ABB RobotStudio station: Celda_Paletizado_20220202-004534.rsstn

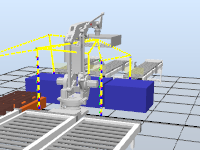
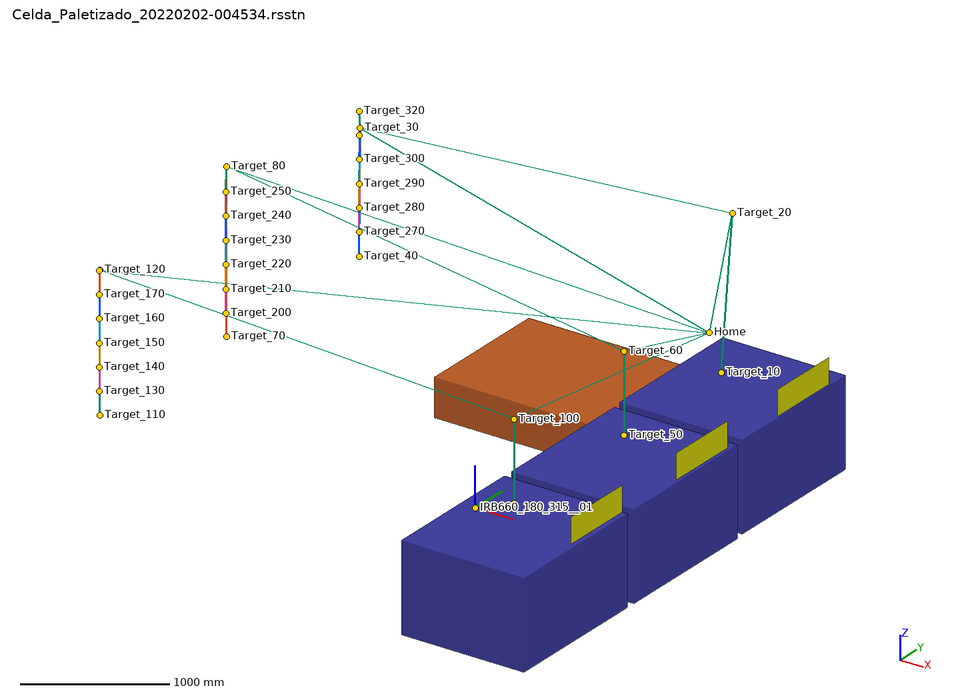
[picture v1: parts stored in the station drawn from their meshes, with robot base, taught points and paths (robot models come from the ABB library and are not in the file)]
Station Celda_Paletizado (saved by RobotStudio 21.4.9700.0)
Controller IRB660_180_315
  mechanical unit ROB_1: IRB660_180_315__01, 6 joints, base frame (0, 0, 0) mm
Layout (positions relative to the parent item):
  - IRB660_180_315__01 [mechanism, from Robots\IRB660_180_315__01.rslib] at (0, 0, 0) mm; joint values [0, 0.0198, -0.194, 0] (rad or m)
  - 600_guide [part, from Equipment\Conveyor Guide 600.rslib] at (4720, 275, 0) mm, rotated rx 0 ry 0 rz 180 deg
  - 600_guide_2 [part, from Equipment\Conveyor Guide 600.rslib] at (4720, 1475, 0) mm, rotated rx 0 ry 0 rz 180 deg
  - 600_guide_3 [part, from Equipment\Conveyor Guide 600.rslib] at (4720, -900, 0) mm, rotated rx 0 ry 0 rz 180 deg
  - 1200_4000_h2_2 [part, from Equipment\Conveyor 1200 4000 h2.rslib] at (-1500, -1000, 0) mm, rotated rx 0 ry 0 rz 180 deg
  - 1200_4000_h2_3 [part, from Equipment\Conveyor 1200 4000 h2.rslib] at (-1500, 2000, 0) mm, rotated rx 0 ry 0 rz 180 deg
  - 1200_4000_h2_4 [part, from Equipment\Conveyor 1200 4000 h2.rslib] at (-1500, 500, 0) mm, rotated rx 0 ry 0 rz 180 deg
  - 1200_4800_h2_2 [part, from Equipment\Conveyor 1200 4800 h2.rslib] at (-6865.5, 2181.45, 0) mm, rotated rx 0 ry 0 rz -90 deg
  - Pieza_1 [part] at (-5740.3, -4363.37, 0) mm, rotated rx 0 ry 0 rz 90 deg, size 1600 x 1000 x 355 mm
  - wraping_1 [part] at (-6239.59, -3461.03, 366.67) mm, rotated rx 0 ry 0 rz -90 deg, size 2370 x 1393.7 x 2100 mm
  - wraping_2 [part] at (-6238.99, -3463.39, 358.4) mm, rotated rx 0 ry 0 rz -90 deg, size 1400 x 1393.6 x 350 mm
  - wraping_3 [part] at (-6242.7, -3445.47, -111.4) mm, rotated rx 90 ry 0 rz -90 deg, size 323.7 x 500 x 658.2 mm
  - Pieza_4 [part] at (-1012.61, 969.79, 0) mm, size 1300 x 1100 x 300 mm
  - Pieza_6 [part] at (689.01, 695.64, 0) mm, size 1000 x 1200 x 700 mm
  - Pieza_7 [part] at (702.6, -1863.75, 0) mm, size 1000 x 1200 x 700 mm
  - Pieza_8 [part] at (703.57, -585.32, 0) mm, size 1000 x 1200 x 700 mm
  - Mi_mecanismo [mechanism] at (1910, 0, 2093) mm; joint values [0, 0] (rad or m)
      TCP Mi_mecanismo_1 at (1.05, 425.12, 399.16) mm, rotated rx 90 ry 0 rz 180 deg
      links: L1, L2, L3
  - Euro Pallet [graphiccomponentgroup, from Equipment\Euro Pallet.rslib] at (223.77, 1878.53, 297.19) mm, rotated rx 0 ry 0 rz 180 deg
    - Body 1 [part, from Equipment\Euro Pallet.rslib]
  - Euro Pallet_2 [graphiccomponentgroup, from Equipment\Euro Pallet.rslib] at (-1565.85, 821.96, 434.35) mm, rotated rx 0 ry 0 rz 90 deg
    - Body 1 [part, from Equipment\Euro Pallet.rslib]
  - Pieza_19 [part] at (1027.44, -3056.32, 715) mm, rotated rx 0 ry 0 rz 90 deg, size 425 x 325 x 180 mm
  - Pequeño [smart component] at (5282.75, -525.09, 765.47) mm
      signals: DI Start, DI Cinta, DI Coger, DI Soltar, DO Sensor1, DO Recoger_peq
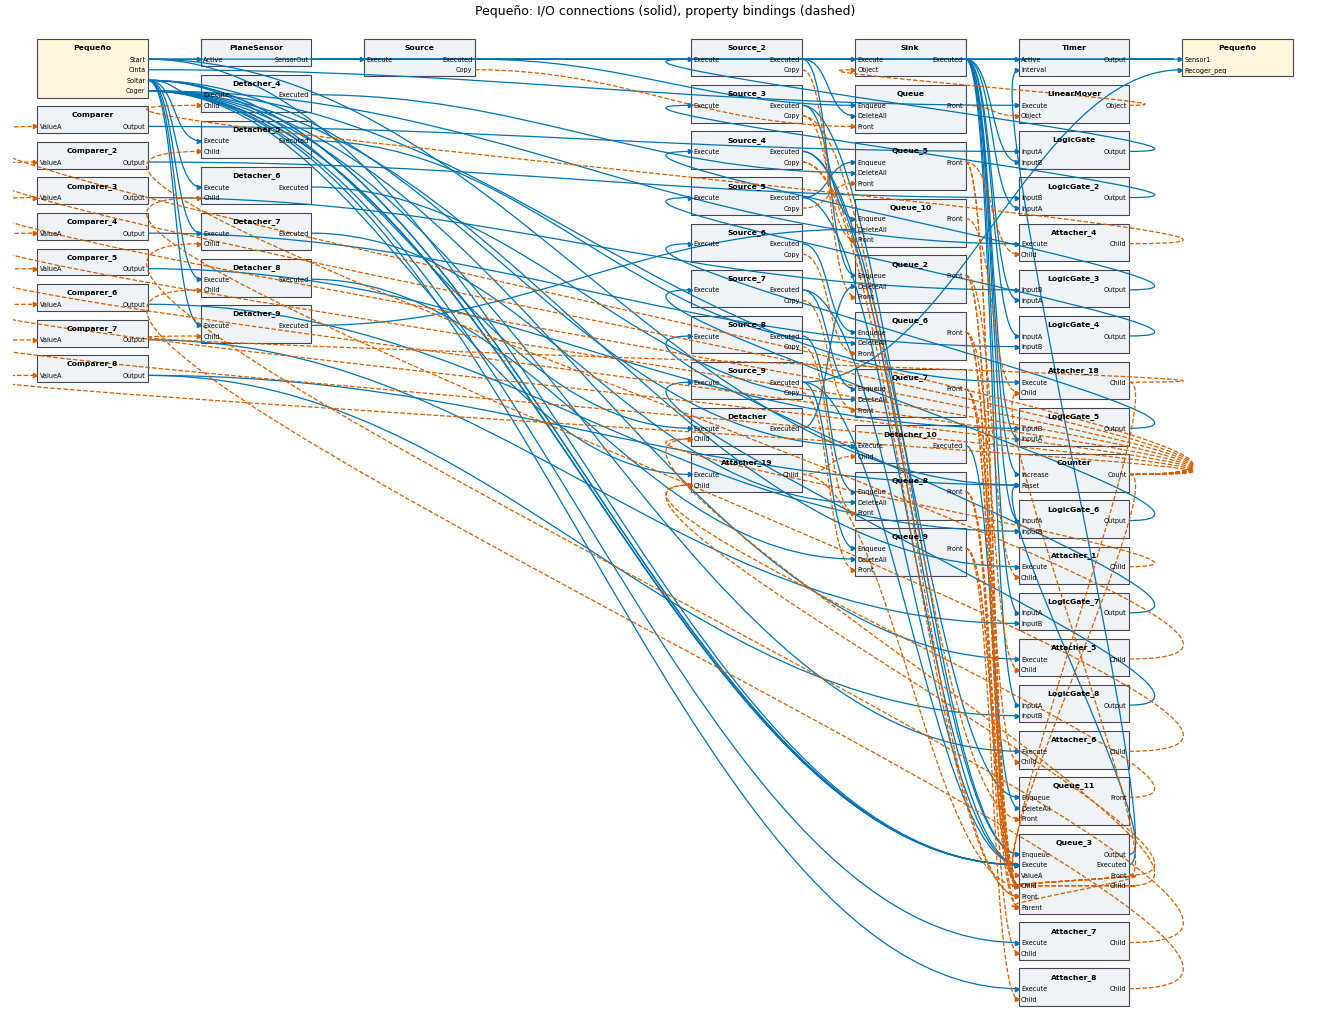
      connections:
        Pequeño.Start -> Timer.Active
        Timer.Output -> Source.Execute
        Source.Executed -> Queue.Enqueue
        Pequeño.Cinta -> LinearMover.Execute
        Pequeño.Start -> PlaneSensor.Active
        PlaneSensor.SensorOut -> Sink.Execute
        Source_2.Executed -> Queue_2.Enqueue
        Sink.Executed -> Counter.Increase
        LogicGate.Output -> Source_2.Execute
        Comparer.Output -> LogicGate.InputA
        Sink.Executed -> LogicGate.InputB
        Comparer_2.Output -> LogicGate_2.InputB
        Sink.Executed -> LogicGate_2.InputA
        LogicGate_2.Output -> Source_3.Execute
        Source_3.Executed -> Queue_3.Enqueue
        PlaneSensor.SensorOut -> Pequeño.Sensor1
        Comparer_3.Output -> LogicGate_3.InputB
        LogicGate_3.Output -> Source_4.Execute
        Sink.Executed -> LogicGate_3.InputA
        Source_4.Executed -> Queue_4.Enqueue
        Sink.Executed -> LogicGate_4.InputA
        Comparer_4.Output -> LogicGate_4.InputB
        LogicGate_4.Output -> Source_5.Execute
        Source_5.Executed -> Queue_5.Enqueue
        Comparer_5.Output -> LogicGate_5.InputB
        Sink.Executed -> LogicGate_5.InputA
        LogicGate_5.Output -> Source_6.Execute
        Source_6.Executed -> Queue_6.Enqueue
        Sink.Executed -> LogicGate_6.InputA
        Comparer_6.Output -> LogicGate_6.InputB
        LogicGate_6.Output -> Source_7.Execute
        Source_7.Executed -> Queue_7.Enqueue
        Sink.Executed -> LogicGate_7.InputA
        Comparer_7.Output -> LogicGate_7.InputB
        LogicGate_7.Output -> Source_8.Execute
        Source_8.Executed -> Queue_8.Enqueue
        Sink.Executed -> LogicGate_8.InputA
        Comparer_8.Output -> LogicGate_8.InputB
        LogicGate_8.Output -> Source_9.Execute
        Source_9.Executed -> Queue_9.Enqueue
        Comparer_9.Output -> Counter.Reset
        Comparer_8.Output -> Counter.Reset
        Pequeño.Start -> Counter.Reset
        Pequeño.Soltar -> Detacher.Execute
        Source_9.Executed -> Pequeño.Recoger_peq
        Pequeño.Coger -> Attacher.Execute
        Source_7.Executed -> Attacher_6.Execute
        Source_5.Executed -> Attacher_5.Execute
        Source_9.Executed -> Attacher_7.Execute
        Pequeño.Coger -> Attacher_1.Execute
        Pequeño.Coger -> Attacher_2.Execute
        Pequeño.Coger -> Attacher_3.Execute
        Pequeño.Coger -> Attacher_4.Execute
        Pequeño.Coger -> Attacher_5.Execute
        Pequeño.Coger -> Attacher_6.Execute
        Pequeño.Coger -> Attacher_7.Execute
        Pequeño.Coger -> Attacher_8.Execute
        Pequeño.Soltar -> Detacher_2.Execute
        Pequeño.Soltar -> Detacher_3.Execute
        Pequeño.Soltar -> Detacher_4.Execute
        Pequeño.Soltar -> Detacher_5.Execute
        Pequeño.Soltar -> Detacher_6.Execute
        Pequeño.Soltar -> Detacher_7.Execute
        Pequeño.Soltar -> Detacher_8.Execute
        Pequeño.Coger -> Attacher_18.Execute
        Pequeño.Coger -> Attacher_19.Execute
        Pequeño.Soltar -> Detacher_9.Execute
        Pequeño.Soltar -> Detacher_10.Execute
        Source_4.Executed -> Queue_11.Enqueue
        Source_3.Executed -> Queue_10.Enqueue
        Source_2.Executed -> Queue.DeleteAll
        Detacher.Executed -> Queue_2.DeleteAll
        Detacher_9.Executed -> Queue_10.DeleteAll
        Detacher_10.Executed -> Queue_11.DeleteAll
        Detacher_4.Executed -> Queue_5.DeleteAll
        Detacher_5.Executed -> Queue_6.DeleteAll
        Detacher_6.Executed -> Queue_7.DeleteAll
        Detacher_7.Executed -> Queue_8.DeleteAll
        Detacher_8.Executed -> Queue_9.DeleteAll
        Random.Executed -> Timer.Interval
        Pequeño.Start -> Random.Execute
        Source.Copy => Queue.Front
        Queue.Front => LinearMover.Object
        LinearMover.Object => Sink.Object
        Counter.Count => Comparer.ValueA
        Counter.Count => Comparer_2.ValueA
        Counter.Count => Comparer_3.ValueA
        Counter.Count => Comparer_4.ValueA
        Counter.Count => Comparer_5.ValueA
        Counter.Count => Comparer_6.ValueA
        Counter.Count => Comparer_7.ValueA
        Counter.Count => Comparer_8.ValueA
        Counter.Count => Comparer_9.ValueA
        Queue_2.Front => Attacher.Child
        Queue_3.Front => Attacher.Child
        Queue_4.Front => Attacher.Child
        Queue_5.Front => Attacher.Child
        Queue_6.Front => Attacher.Child
        Queue_7.Front => Attacher.Child
        Queue_8.Front => Attacher.Child
        Queue_9.Front => Attacher.Child
        Attacher.Child => Detacher.Child
        Source_2.Copy => Queue_2.Front
        Source_3.Copy => Queue_3.Front
        Source_4.Copy => Queue_4.Front
        Source_5.Copy => Queue_5.Front
        Source_6.Copy => Queue_6.Front
        Source_7.Copy => Queue_7.Front
        Source_8.Copy => Queue_8.Front
        Source_9.Copy => Queue_9.Front
        Queue_2.Front => Attacher_3.Child
        Attacher_1.Child => Detacher.Child
        Queue_4.Front => Attacher_5.Parent
        Queue_5.Front => Attacher_5.Child
        Queue_6.Front => Attacher_6.Parent
        Queue_7.Front => Attacher_6.Child
        Queue_8.Front => Attacher_7.Parent
        Queue_9.Front => Attacher_7.Child
        Queue_3.Front => Attacher_2.Child
        Queue_4.Front => Attacher_3.Child
        Queue_5.Front => Attacher_4.Child
        Queue_6.Front => Attacher_5.Child
        Queue_7.Front => Attacher_6.Child
        Queue_8.Front => Attacher_7.Child
        Queue_9.Front => Attacher_8.Child
        Attacher_2.Child => Detacher_2.Child
        Attacher_3.Child => Detacher_3.Child
        Attacher_4.Child => Detacher_4.Child
        Attacher_5.Child => Detacher_5.Child
        Attacher_6.Child => Detacher_6.Child
        Attacher_7.Child => Detacher_7.Child
        Attacher_8.Child => Detacher_8.Child
        Queue_2.Front => Attacher_1.Child
        Queue_3.Front => Attacher_18.Child
        Queue_4.Front => Attacher_19.Child
        Attacher_18.Child => Detacher_2.Child
        Attacher_19.Child => Detacher_3.Child
        Source_4.Copy => Queue_11.Front
        Source_3.Copy => Queue_10.Front
        Queue_10.Front => Attacher_18.Child
        Queue_11.Front => Attacher_19.Child
        Attacher_18.Child => Detacher_9.Child
        Attacher_19.Child => Detacher_10.Child
    - LinearMover [smart component, from Components\LinearMover.rslib]
        properties: Object=(none); Direction=[-0.001 0 0]; Speed=1.5; Reference=Global; ReferenceObject=(none)
    - PlaneSensor [smart component, from Components\PlaneSensor.rslib] at (-3443.45, 1412.3, 72.76) mm, rotated rx 0 ry -90 rz 0 deg
        properties: Origin=[0 0 0]; Axis1=[0.2 0 0]; Axis2=[0 0.6 0]; SensedPart=(none)
      - _sensorPart_ [part], size 200 x 600 x 0 mm
    - Detacher [smart component, from Components\Detacher.rslib]
        properties: Child=(none); KeepPosition=true
    - Queue [smart component, from Components\Queue.rslib]
        properties: Back=(none); Front=(none); Queue=; NumberOfObjects=0
    - Source [smart component, from Components\Source.rslib]
        properties: Source=Pieza_19; Copy=(none); Parent=(none); Position=[4.6 0.975 0.775]; Orientation=[0 0 1.5707963267949]; Transient=true; PhysicsBehavior=0
    - Timer [smart component, from Components\Timer.rslib]
        properties: StartTime=0; Interval=3; Repeat=true; CurrentTime=11.448
    - Sink [smart component, from Components\Sink.rslib]
        properties: Object=(none)
    - Source_2 [smart component, from Components\Source.rslib]
        properties: Source=Pieza_19; Copy=(none); Parent=(none); Position=[1.015 1.47 0.7]; Orientation=[0 0 1.5707963267949]; Transient=false; PhysicsBehavior=0
    - Source_3 [smart component, from Components\Source.rslib]
        properties: Source=Pieza_19; Copy=(none); Parent=(none); Position=[1.345 1.47 0.7]; Orientation=[0 0 1.5707963267949]; Transient=false; PhysicsBehavior=0
    - Source_4 [smart component, from Components\Source.rslib]
        properties: Source=Pieza_19; Copy=(none); Parent=(none); Position=[1.675 1.47 0.7]; Orientation=[0 0 1.5707963267949]; Transient=false; PhysicsBehavior=0
    - Queue_2 [smart component, from Components\Queue.rslib]
        properties: Back=(none); Front=(none); Queue=; NumberOfObjects=0
    - Counter [smart component, from Components\Counter.rslib]
        properties: Count=0
    - LogicGate [smart component, from Components\LogicGate.rslib]
        properties: Operator=AND; Delay=0
    - Comparer [smart component, from Components\Comparer.rslib]
        properties: ValueA=0; Operator===; ValueB=1
    - Comparer_2 [smart component, from Components\Comparer.rslib]
        properties: ValueA=0; Operator===; ValueB=2
    - Comparer_3 [smart component, from Components\Comparer.rslib]
        properties: ValueA=0; Operator===; ValueB=3
    - Comparer_4 [smart component, from Components\Comparer.rslib]
        properties: ValueA=0; Operator===; ValueB=4
    - Comparer_5 [smart component, from Components\Comparer.rslib]
        properties: ValueA=0; Operator===; ValueB=5
    - Comparer_6 [smart component, from Components\Comparer.rslib]
        properties: ValueA=0; Operator===; ValueB=6
    - Comparer_7 [smart component, from Components\Comparer.rslib]
        properties: ValueA=0; Operator===; ValueB=7
    - LogicGate_2 [smart component, from Components\LogicGate.rslib]
        properties: Operator=AND; Delay=0
    - LogicGate_3 [smart component, from Components\LogicGate.rslib]
        properties: Operator=AND; Delay=0
    - LogicGate_4 [smart component, from Components\LogicGate.rslib]
        properties: Operator=AND; Delay=0
    - LogicGate_5 [smart component, from Components\LogicGate.rslib]
        properties: Operator=AND; Delay=0
    - LogicGate_6 [smart component, from Components\LogicGate.rslib]
        properties: Operator=AND; Delay=0
    - LogicGate_7 [smart component, from Components\LogicGate.rslib]
        properties: Operator=AND; Delay=0
    - Queue_5 [smart component, from Components\Queue.rslib]
        properties: Back=(none); Front=(none); Queue=; NumberOfObjects=0
    - Queue_6 [smart component, from Components\Queue.rslib]
        properties: Back=(none); Front=(none); Queue=; NumberOfObjects=0
    - Queue_7 [smart component, from Components\Queue.rslib]
        properties: Back=(none); Front=(none); Queue=; NumberOfObjects=0
    - Queue_8 [smart component, from Components\Queue.rslib]
        properties: Back=(none); Front=(none); Queue=; NumberOfObjects=0
    - Source_5 [smart component, from Components\Source.rslib]
        properties: Source=Pieza_19; Copy=(none); Parent=(none); Position=[0.69 1.14 0.7]; Orientation=[0 0 0]; Transient=false; PhysicsBehavior=0
    - Source_6 [smart component, from Components\Source.rslib]
        properties: Source=Pieza_19; Copy=(none); Parent=(none); Position=[1.255 1.14 0.7]; Orientation=[0 0 0]; Transient=false; PhysicsBehavior=0
    - Source_7 [smart component, from Components\Source.rslib]
        properties: Source=Pieza_19; Copy=(none); Parent=(none); Position=[1.015 0.71 0.7]; Orientation=[0 0 1.5707963267949]; Transient=false; PhysicsBehavior=0
    - Source_8 [smart component, from Components\Source.rslib]
        properties: Source=Pieza_19; Copy=(none); Parent=(none); Position=[1.345 0.71 0.7]; Orientation=[0 0 1.5707963267949]; Transient=false; PhysicsBehavior=0
    - Comparer_8 [smart component, from Components\Comparer.rslib]
        properties: ValueA=0; Operator=>=; ValueB=8
    - Source_9 [smart component, from Components\Source.rslib]
        properties: Source=Pieza_19; Copy=(none); Parent=(none); Position=[1.675 0.71 0.7]; Orientation=[0 0 1.5707963267949]; Transient=false; PhysicsBehavior=0
    - Queue_9 [smart component, from Components\Queue.rslib]
        properties: Back=(none); Front=(none); Queue=; NumberOfObjects=0
    - LogicGate_8 [smart component, from Components\LogicGate.rslib]
        properties: Operator=AND; Delay=0
    - Attacher_1 [smart component, from Components\Attacher.rslib]
        properties: Parent=Mi_mecanismo; Flange=0; Child=(none); Mount=false; Offset=[0 0 0]; Orientation=[0 0 0]
    - Attacher_4 [smart component, from Components\Attacher.rslib]
        properties: Parent=Mi_mecanismo; Flange=0; Child=(none); Mount=false; Offset=[0 0 0]; Orientation=[0 0 0]
    - Attacher_5 [smart component, from Components\Attacher.rslib]
        properties: Parent=Mi_mecanismo; Flange=0; Child=(none); Mount=false; Offset=[0 0 0]; Orientation=[0 0 0]
    - Attacher_6 [smart component, from Components\Attacher.rslib]
        properties: Parent=Mi_mecanismo; Flange=0; Child=(none); Mount=false; Offset=[0 0 0]; Orientation=[0 0 0]
    - Attacher_7 [smart component, from Components\Attacher.rslib]
        properties: Parent=Mi_mecanismo; Flange=0; Child=(none); Mount=false; Offset=[0 0 0]; Orientation=[0 0 0]
    - Attacher_8 [smart component, from Components\Attacher.rslib]
        properties: Parent=Mi_mecanismo; Flange=0; Child=(none); Mount=false; Offset=[0 0 0]; Orientation=[0 0 0]
    - Detacher_4 [smart component, from Components\Detacher.rslib]
        properties: Child=(none); KeepPosition=true
    - Detacher_5 [smart component, from Components\Detacher.rslib]
        properties: Child=(none); KeepPosition=true
    - Detacher_6 [smart component, from Components\Detacher.rslib]
        properties: Child=(none); KeepPosition=true
    - Detacher_7 [smart component, from Components\Detacher.rslib]
        properties: Child=(none); KeepPosition=true
    - Detacher_8 [smart component, from Components\Detacher.rslib]
        properties: Child=(none); KeepPosition=true
    - Attacher_18 [smart component, from Components\Attacher.rslib]
        properties: Parent=Mi_mecanismo; Flange=0; Child=(none); Mount=false; Offset=[0 0 0]; Orientation=[0 0 0]
    - Attacher_19 [smart component, from Components\Attacher.rslib]
        properties: Parent=Mi_mecanismo; Flange=0; Child=(none); Mount=false; Offset=[0 0 0]; Orientation=[0 0 0]
    - Detacher_9 [smart component, from Components\Detacher.rslib]
        properties: Child=(none); KeepPosition=true
    - Detacher_10 [smart component, from Components\Detacher.rslib]
        properties: Child=(none); KeepPosition=true
    - Queue_10 [smart component, from Components\Queue.rslib]
        properties: Back=(none); Front=(none); Queue=; NumberOfObjects=0
    - Queue_11 [smart component, from Components\Queue.rslib]
        properties: Back=(none); Front=(none); Queue=; NumberOfObjects=0
  - Pallet [smart component]
      signals: DI Start_pallet
      connections:
        Pallet.Start_pallet -> LogicGate_10.InputA
        Pallet.Start_pallet -> PlaneSensor.Active
        PlaneSensor.SensorOut -> LogicGate_10.InputB
    - LogicGate_10 [smart component, from Components\LogicGate.rslib]
        properties: Operator=AND; Delay=0
    - Queue_10 [smart component, from Components\Queue.rslib]
        properties: Back=(none); Front=(none); Queue=; NumberOfObjects=0
    - Source_10 [smart component, from Components\Source.rslib]
        properties: Source=(none); Copy=(none); Parent=(none); Position=[0 0 0]; Orientation=[0 0 0]; Transient=false; PhysicsBehavior=0
    - Comparer_10 [smart component, from Components\Comparer.rslib]
        properties: ValueA=0; Operator===; ValueB=0
    - Counter [smart component, from Components\Counter.rslib]
        properties: Count=0
    - Sink [smart component, from Components\Sink.rslib]
        properties: Object=(none)
    - PlaneSensor [smart component, from Components\PlaneSensor.rslib]
        properties: Origin=[0 0 0]; Axis1=[0.1 0 0]; Axis2=[0 0.1 0]; SensedPart=(none)
      - _sensorPart_ [part, from Components\PlaneSensor.rslib]
    - PlaneSensor_2 [smart component, from Components\PlaneSensor.rslib]
        properties: Origin=[0 0 0]; Axis1=[0.1 0 0]; Axis2=[0 0.1 0]; SensedPart=(none)
      - _sensorPart_ [part, from Components\PlaneSensor.rslib]
    - PlaneSensor_3 [smart component, from Components\PlaneSensor.rslib]
        properties: Origin=[0 0 0]; Axis1=[0.1 0 0]; Axis2=[0 0.1 0]; SensedPart=(none)
      - _sensorPart_ [part, from Components\PlaneSensor.rslib]
    - PlaneSensor_4 [smart component, from Components\PlaneSensor.rslib]
        properties: Origin=[0 0 0]; Axis1=[0.1 0 0]; Axis2=[0 0.1 0]; SensedPart=(none)
      - _sensorPart_ [part, from Components\PlaneSensor.rslib]
    - Attacher [smart component, from Components\Attacher.rslib]
        properties: Parent=(none); Flange=0; Child=(none); Mount=false; Offset=[0 0 0]; Orientation=[0 0 0]
    - Detacher [smart component, from Components\Detacher.rslib]
        properties: Child=(none); KeepPosition=true
    - LinearMover [smart component, from Components\LinearMover.rslib]
        properties: Object=(none); Direction=[1 0 0]; Speed=0; Reference=Global; ReferenceObject=(none)
  - Grande [smart component]
      signals: DI Start, DI Cinta, DI Coger, DI Soltar, DO Sensor1, DO Recoger_peq
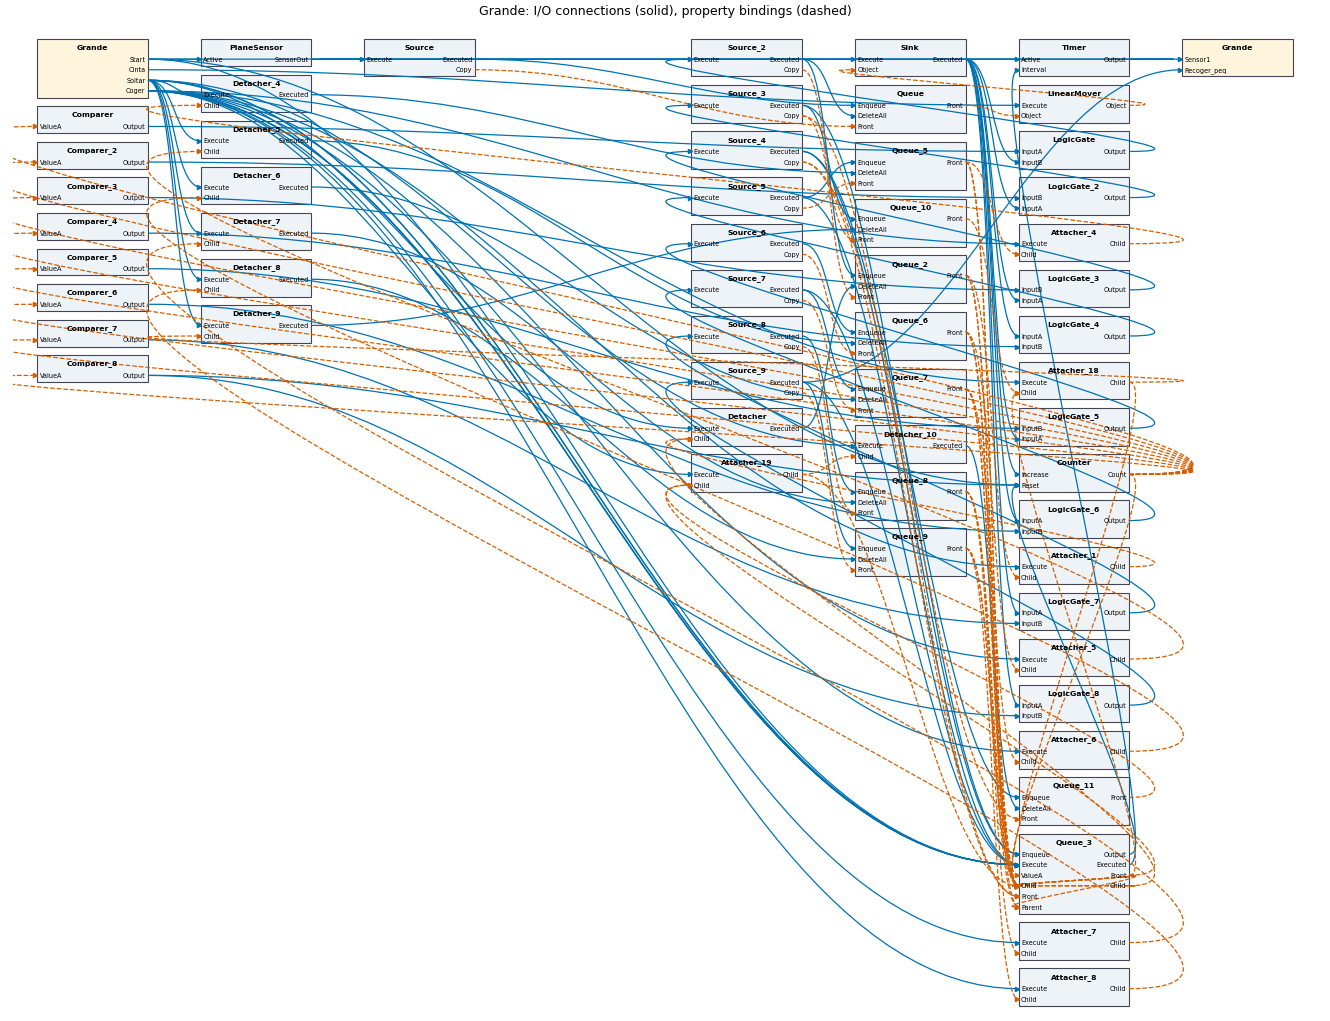
      connections:
        Grande.Start -> Timer.Active
        Timer.Output -> Source.Execute
        Source.Executed -> Queue.Enqueue
        Grande.Cinta -> LinearMover.Execute
        Grande.Start -> PlaneSensor.Active
        PlaneSensor.SensorOut -> Sink.Execute
        Source_2.Executed -> Queue_2.Enqueue
        Sink.Executed -> Counter.Increase
        LogicGate.Output -> Source_2.Execute
        Comparer.Output -> LogicGate.InputA
        Sink.Executed -> LogicGate.InputB
        Comparer_2.Output -> LogicGate_2.InputB
        Sink.Executed -> LogicGate_2.InputA
        LogicGate_2.Output -> Source_3.Execute
        Source_3.Executed -> Queue_3.Enqueue
        PlaneSensor.SensorOut -> Grande.Sensor1
        Comparer_3.Output -> LogicGate_3.InputB
        LogicGate_3.Output -> Source_4.Execute
        Sink.Executed -> LogicGate_3.InputA
        Source_4.Executed -> Queue_4.Enqueue
        Sink.Executed -> LogicGate_4.InputA
        Comparer_4.Output -> LogicGate_4.InputB
        LogicGate_4.Output -> Source_5.Execute
        Source_5.Executed -> Queue_5.Enqueue
        Comparer_5.Output -> LogicGate_5.InputB
        Sink.Executed -> LogicGate_5.InputA
        LogicGate_5.Output -> Source_6.Execute
        Source_6.Executed -> Queue_6.Enqueue
        Sink.Executed -> LogicGate_6.InputA
        Comparer_6.Output -> LogicGate_6.InputB
        LogicGate_6.Output -> Source_7.Execute
        Source_7.Executed -> Queue_7.Enqueue
        Sink.Executed -> LogicGate_7.InputA
        Comparer_7.Output -> LogicGate_7.InputB
        LogicGate_7.Output -> Source_8.Execute
        Source_8.Executed -> Queue_8.Enqueue
        Sink.Executed -> LogicGate_8.InputA
        Comparer_8.Output -> LogicGate_8.InputB
        LogicGate_8.Output -> Source_9.Execute
        Source_9.Executed -> Queue_9.Enqueue
        ?.Output -> Counter.Reset
        Comparer_8.Output -> Counter.Reset
        Grande.Start -> Counter.Reset
        Grande.Soltar -> Detacher.Execute
        Source_9.Executed -> Grande.Recoger_peq
        Grande.Coger -> Attacher.Execute
        Source_7.Executed -> Attacher_6.Execute
        Source_5.Executed -> Attacher_5.Execute
        Source_9.Executed -> Attacher_7.Execute
        Grande.Coger -> Attacher_1.Execute
        Grande.Coger -> Attacher_2.Execute
        Grande.Coger -> Attacher_3.Execute
        Grande.Coger -> Attacher_4.Execute
        Grande.Coger -> Attacher_5.Execute
        Grande.Coger -> Attacher_6.Execute
        Grande.Coger -> Attacher_7.Execute
        Grande.Coger -> Attacher_8.Execute
        Grande.Soltar -> Detacher_2.Execute
        Grande.Soltar -> Detacher_3.Execute
        Grande.Soltar -> Detacher_4.Execute
        Grande.Soltar -> Detacher_5.Execute
        Grande.Soltar -> Detacher_6.Execute
        Grande.Soltar -> Detacher_7.Execute
        Grande.Soltar -> Detacher_8.Execute
        Grande.Coger -> Attacher_18.Execute
        Grande.Coger -> Attacher_19.Execute
        Grande.Soltar -> Detacher_9.Execute
        Grande.Soltar -> Detacher_10.Execute
        Source_4.Executed -> Queue_11.Enqueue
        Source_3.Executed -> Queue_10.Enqueue
        Source_2.Executed -> Queue.DeleteAll
        Detacher.Executed -> Queue_2.DeleteAll
        Detacher_9.Executed -> Queue_10.DeleteAll
        Detacher_10.Executed -> Queue_11.DeleteAll
        Detacher_4.Executed -> Queue_5.DeleteAll
        Detacher_5.Executed -> Queue_6.DeleteAll
        Detacher_6.Executed -> Queue_7.DeleteAll
        Detacher_7.Executed -> Queue_8.DeleteAll
        Detacher_8.Executed -> Queue_9.DeleteAll
        Random_3.Executed -> Timer.Interval
        Grande.Start -> Random_3.Execute
        Source.Copy => Queue.Front
        Queue.Front => LinearMover.Object
        LinearMover.Object => Sink.Object
        Counter.Count => Comparer.ValueA
        Counter.Count => Comparer_2.ValueA
        Counter.Count => Comparer_3.ValueA
        Counter.Count => Comparer_4.ValueA
        Counter.Count => Comparer_5.ValueA
        Counter.Count => Comparer_6.ValueA
        Counter.Count => Comparer_7.ValueA
        Counter.Count => Comparer_8.ValueA
        Counter.Count => ?.ValueA
        Queue_2.Front => Attacher.Child
        Queue_3.Front => Attacher.Child
        Queue_4.Front => Attacher.Child
        Queue_5.Front => Attacher.Child
        Queue_6.Front => Attacher.Child
        Queue_7.Front => Attacher.Child
        Queue_8.Front => Attacher.Child
        Queue_9.Front => Attacher.Child
        Attacher.Child => Detacher.Child
        Source_2.Copy => Queue_2.Front
        Source_3.Copy => Queue_3.Front
        Source_4.Copy => Queue_4.Front
        Source_5.Copy => Queue_5.Front
        Source_6.Copy => Queue_6.Front
        Source_7.Copy => Queue_7.Front
        Source_8.Copy => Queue_8.Front
        Source_9.Copy => Queue_9.Front
        Queue_2.Front => Attacher_3.Child
        Attacher_1.Child => Detacher.Child
        Queue_4.Front => Attacher_5.Parent
        Queue_5.Front => Attacher_5.Child
        Queue_6.Front => Attacher_6.Parent
        Queue_7.Front => Attacher_6.Child
        Queue_8.Front => Attacher_7.Parent
        Queue_9.Front => Attacher_7.Child
        Queue_3.Front => Attacher_2.Child
        Queue_4.Front => Attacher_3.Child
        Queue_5.Front => Attacher_4.Child
        Queue_6.Front => Attacher_5.Child
        Queue_7.Front => Attacher_6.Child
        Queue_8.Front => Attacher_7.Child
        Queue_9.Front => Attacher_8.Child
        Attacher_2.Child => Detacher_2.Child
        Attacher_3.Child => Detacher_3.Child
        Attacher_4.Child => Detacher_4.Child
        Attacher_5.Child => Detacher_5.Child
        Attacher_6.Child => Detacher_6.Child
        Attacher_7.Child => Detacher_7.Child
        Attacher_8.Child => Detacher_8.Child
        Queue_2.Front => Attacher_1.Child
        Queue_3.Front => Attacher_18.Child
        Queue_4.Front => Attacher_19.Child
        Attacher_18.Child => Detacher_2.Child
        Attacher_19.Child => Detacher_3.Child
        Source_4.Copy => Queue_11.Front
        Source_3.Copy => Queue_10.Front
        Queue_10.Front => Attacher_18.Child
        Queue_11.Front => Attacher_19.Child
        Attacher_18.Child => Detacher_9.Child
        Attacher_19.Child => Detacher_10.Child
    - LinearMover [smart component, from Components\LinearMover.rslib]
        properties: Object=(none); Direction=[-0.001 0 0]; Speed=1.5; Reference=Global; ReferenceObject=(none)
    - PlaneSensor [smart component, from Components\PlaneSensor.rslib] at (1833.87, -1506.89, 845.2) mm, rotated rx 0 ry -90 rz 0 deg
        properties: Origin=[0 0 0]; Axis1=[0.2 0 0]; Axis2=[0 0.6 0]; SensedPart=(none)
      - _sensorPart_ [part], size 200 x 600 x 0 mm
    - Detacher [smart component, from Components\Detacher.rslib]
        properties: Child=(none); KeepPosition=true
    - Queue [smart component, from Components\Queue.rslib]
        properties: Back=(none); Front=(none); Queue=; NumberOfObjects=0
    - Source [smart component, from Components\Source.rslib]
        properties: Source=Pieza_19; Copy=(none); Parent=(none); Position=[4.6 -1.595 0.775]; Orientation=[0 0 1.5707963267949]; Transient=true; PhysicsBehavior=0
    - Timer [smart component, from Components\Timer.rslib]
        properties: StartTime=0; Interval=5; Repeat=true; CurrentTime=11.448
    - Sink [smart component, from Components\Sink.rslib]
        properties: Object=(none)
    - Source_2 [smart component, from Components\Source.rslib]
        properties: Source=Pieza_19; Copy=(none); Parent=(none); Position=[1.015 -1.1 0.7]; Orientation=[0 0 1.5707963267949]; Transient=false; PhysicsBehavior=0
    - Source_3 [smart component, from Components\Source.rslib]
        properties: Source=Pieza_19; Copy=(none); Parent=(none); Position=[1.345 -1.1 0.7]; Orientation=[0 0 1.5707963267949]; Transient=false; PhysicsBehavior=0
    - Source_4 [smart component, from Components\Source.rslib]
        properties: Source=Pieza_19; Copy=(none); Parent=(none); Position=[1.675 -1.1 0.7]; Orientation=[0 0 1.5707963267949]; Transient=false; PhysicsBehavior=0
    - Queue_2 [smart component, from Components\Queue.rslib]
        properties: Back=(none); Front=(none); Queue=; NumberOfObjects=0
    - Counter [smart component, from Components\Counter.rslib]
        properties: Count=0
    - LogicGate [smart component, from Components\LogicGate.rslib]
        properties: Operator=AND; Delay=0
    - Comparer [smart component, from Components\Comparer.rslib]
        properties: ValueA=0; Operator===; ValueB=1
    - Comparer_2 [smart component, from Components\Comparer.rslib]
        properties: ValueA=0; Operator===; ValueB=2
    - Comparer_3 [smart component, from Components\Comparer.rslib]
        properties: ValueA=0; Operator===; ValueB=3
    - Comparer_4 [smart component, from Components\Comparer.rslib]
        properties: ValueA=0; Operator===; ValueB=4
    - Comparer_5 [smart component, from Components\Comparer.rslib]
        properties: ValueA=0; Operator===; ValueB=5
    - Comparer_6 [smart component, from Components\Comparer.rslib]
        properties: ValueA=0; Operator===; ValueB=6
    - Comparer_7 [smart component, from Components\Comparer.rslib]
        properties: ValueA=0; Operator===; ValueB=7
    - LogicGate_2 [smart component, from Components\LogicGate.rslib]
        properties: Operator=AND; Delay=0
    - LogicGate_3 [smart component, from Components\LogicGate.rslib]
        properties: Operator=AND; Delay=0
    - LogicGate_4 [smart component, from Components\LogicGate.rslib]
        properties: Operator=AND; Delay=0
    - LogicGate_5 [smart component, from Components\LogicGate.rslib]
        properties: Operator=AND; Delay=0
    - LogicGate_6 [smart component, from Components\LogicGate.rslib]
        properties: Operator=AND; Delay=0
    - LogicGate_7 [smart component, from Components\LogicGate.rslib]
        properties: Operator=AND; Delay=0
    - Queue_5 [smart component, from Components\Queue.rslib]
        properties: Back=(none); Front=(none); Queue=; NumberOfObjects=0
    - Queue_6 [smart component, from Components\Queue.rslib]
        properties: Back=(none); Front=(none); Queue=; NumberOfObjects=0
    - Queue_7 [smart component, from Components\Queue.rslib]
        properties: Back=(none); Front=(none); Queue=; NumberOfObjects=0
    - Queue_8 [smart component, from Components\Queue.rslib]
        properties: Back=(none); Front=(none); Queue=; NumberOfObjects=0
    - Source_5 [smart component, from Components\Source.rslib]
        properties: Source=Pieza_19; Copy=(none); Parent=(none); Position=[0.69 -1.43 0.7]; Orientation=[0 0 0]; Transient=false; PhysicsBehavior=0
    - Source_6 [smart component, from Components\Source.rslib]
        properties: Source=Pieza_19; Copy=(none); Parent=(none); Position=[1.255 -1.43 0.7]; Orientation=[0 0 0]; Transient=false; PhysicsBehavior=0
    - Source_7 [smart component, from Components\Source.rslib]
        properties: Source=Pieza_19; Copy=(none); Parent=(none); Position=[1.015 -1.86 0.7]; Orientation=[0 0 1.5707963267949]; Transient=false; PhysicsBehavior=0
    - Source_8 [smart component, from Components\Source.rslib]
        properties: Source=Pieza_19; Copy=(none); Parent=(none); Position=[1.345 -1.86 0.7]; Orientation=[0 0 1.5707963267949]; Transient=false; PhysicsBehavior=0
    - Comparer_8 [smart component, from Components\Comparer.rslib]
        properties: ValueA=0; Operator=>=; ValueB=8
    - Source_9 [smart component, from Components\Source.rslib]
        properties: Source=Pieza_19; Copy=(none); Parent=(none); Position=[1.675 -1.86 0.7]; Orientation=[0 0 1.5707963267949]; Transient=false; PhysicsBehavior=0
    - Queue_9 [smart component, from Components\Queue.rslib]
        properties: Back=(none); Front=(none); Queue=; NumberOfObjects=0
    - LogicGate_8 [smart component, from Components\LogicGate.rslib]
        properties: Operator=AND; Delay=0
    - Attacher_1 [smart component, from Components\Attacher.rslib]
        properties: Parent=Mi_mecanismo; Flange=0; Child=(none); Mount=false; Offset=[0 0 0]; Orientation=[0 0 0]
    - Attacher_4 [smart component, from Components\Attacher.rslib]
        properties: Parent=Mi_mecanismo; Flange=0; Child=(none); Mount=false; Offset=[0 0 0]; Orientation=[0 0 0]
    - Attacher_5 [smart component, from Components\Attacher.rslib]
        properties: Parent=Mi_mecanismo; Flange=0; Child=(none); Mount=false; Offset=[0 0 0]; Orientation=[0 0 0]
    - Attacher_6 [smart component, from Components\Attacher.rslib]
        properties: Parent=Mi_mecanismo; Flange=0; Child=(none); Mount=false; Offset=[0 0 0]; Orientation=[0 0 0]
    - Attacher_7 [smart component, from Components\Attacher.rslib]
        properties: Parent=Mi_mecanismo; Flange=0; Child=(none); Mount=false; Offset=[0 0 0]; Orientation=[0 0 0]
    - Attacher_8 [smart component, from Components\Attacher.rslib]
        properties: Parent=Mi_mecanismo; Flange=0; Child=(none); Mount=false; Offset=[0 0 0]; Orientation=[0 0 0]
    - Detacher_4 [smart component, from Components\Detacher.rslib]
        properties: Child=(none); KeepPosition=true
    - Detacher_5 [smart component, from Components\Detacher.rslib]
        properties: Child=(none); KeepPosition=true
    - Detacher_6 [smart component, from Components\Detacher.rslib]
        properties: Child=(none); KeepPosition=true
    - Detacher_7 [smart component, from Components\Detacher.rslib]
        properties: Child=(none); KeepPosition=true
    - Detacher_8 [smart component, from Components\Detacher.rslib]
        properties: Child=(none); KeepPosition=true
    - Attacher_18 [smart component, from Components\Attacher.rslib]
        properties: Parent=Mi_mecanismo; Flange=0; Child=(none); Mount=false; Offset=[0 0 0]; Orientation=[0 0 0]
    - Attacher_19 [smart component, from Components\Attacher.rslib]
        properties: Parent=Mi_mecanismo; Flange=0; Child=(none); Mount=false; Offset=[0 0 0]; Orientation=[0 0 0]
    - Detacher_9 [smart component, from Components\Detacher.rslib]
        properties: Child=(none); KeepPosition=true
    - Detacher_10 [smart component, from Components\Detacher.rslib]
        properties: Child=(none); KeepPosition=true
    - Queue_10 [smart component, from Components\Queue.rslib]
        properties: Back=(none); Front=(none); Queue=; NumberOfObjects=0
    - Queue_11 [smart component, from Components\Queue.rslib]
        properties: Back=(none); Front=(none); Queue=; NumberOfObjects=0
  - Mediano [smart component] at (4162.28, 543.28, 0) mm
      signals: DI Start, DI Cinta, DI Coger, DI Soltar, DO Sensor1, DO Recoger_med
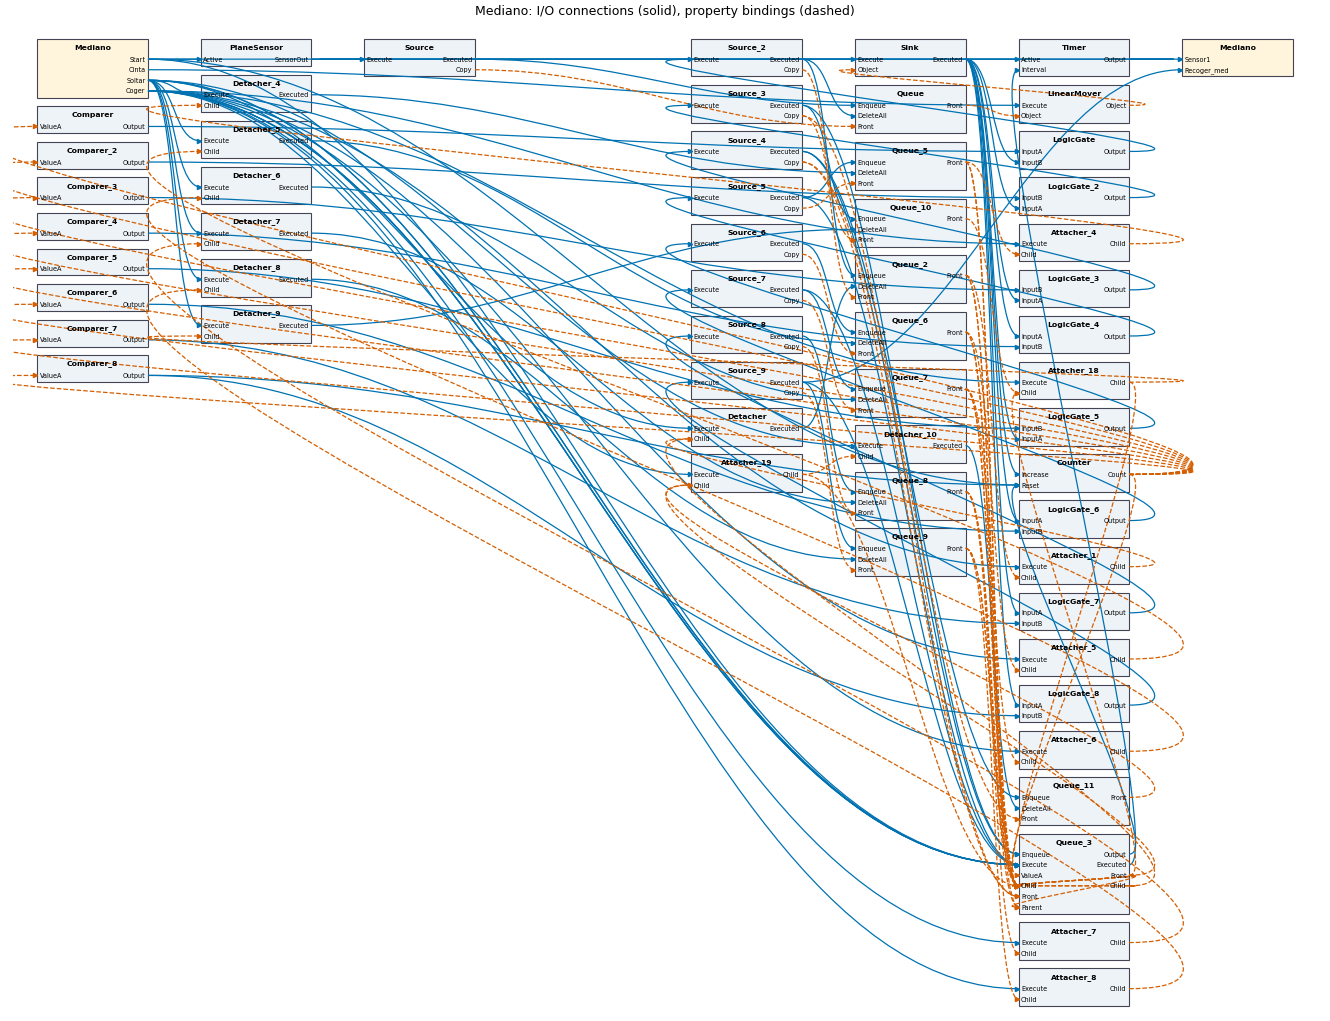
      connections:
        Mediano.Start -> Timer.Active
        Timer.Output -> Source.Execute
        Source.Executed -> Queue.Enqueue
        Mediano.Cinta -> LinearMover.Execute
        Mediano.Start -> PlaneSensor.Active
        PlaneSensor.SensorOut -> Sink.Execute
        Source_2.Executed -> Queue_2.Enqueue
        Sink.Executed -> Counter.Increase
        LogicGate.Output -> Source_2.Execute
        Comparer.Output -> LogicGate.InputA
        Sink.Executed -> LogicGate.InputB
        Comparer_2.Output -> LogicGate_2.InputB
        Sink.Executed -> LogicGate_2.InputA
        LogicGate_2.Output -> Source_3.Execute
        Source_3.Executed -> Queue_3.Enqueue
        PlaneSensor.SensorOut -> Mediano.Sensor1
        Comparer_3.Output -> LogicGate_3.InputB
        LogicGate_3.Output -> Source_4.Execute
        Sink.Executed -> LogicGate_3.InputA
        Source_4.Executed -> Queue_4.Enqueue
        Sink.Executed -> LogicGate_4.InputA
        Comparer_4.Output -> LogicGate_4.InputB
        LogicGate_4.Output -> Source_5.Execute
        Source_5.Executed -> Queue_5.Enqueue
        Comparer_5.Output -> LogicGate_5.InputB
        Sink.Executed -> LogicGate_5.InputA
        LogicGate_5.Output -> Source_6.Execute
        Source_6.Executed -> Queue_6.Enqueue
        Sink.Executed -> LogicGate_6.InputA
        Comparer_6.Output -> LogicGate_6.InputB
        LogicGate_6.Output -> Source_7.Execute
        Source_7.Executed -> Queue_7.Enqueue
        Sink.Executed -> LogicGate_7.InputA
        Comparer_7.Output -> LogicGate_7.InputB
        LogicGate_7.Output -> Source_8.Execute
        Source_8.Executed -> Queue_8.Enqueue
        Sink.Executed -> LogicGate_8.InputA
        Comparer_8.Output -> LogicGate_8.InputB
        LogicGate_8.Output -> Source_9.Execute
        Source_9.Executed -> Queue_9.Enqueue
        ?.Output -> Counter.Reset
        Comparer_8.Output -> Counter.Reset
        Mediano.Start -> Counter.Reset
        Mediano.Soltar -> Detacher.Execute
        Mediano.Coger -> Attacher.Execute
        Source_7.Executed -> Attacher_6.Execute
        Source_5.Executed -> Attacher_5.Execute
        Source_9.Executed -> Attacher_7.Execute
        Mediano.Coger -> Attacher_1.Execute
        Mediano.Coger -> Attacher_2.Execute
        Mediano.Coger -> Attacher_3.Execute
        Mediano.Coger -> Attacher_4.Execute
        Mediano.Coger -> Attacher_5.Execute
        Mediano.Coger -> Attacher_6.Execute
        Mediano.Coger -> Attacher_7.Execute
        Mediano.Coger -> Attacher_8.Execute
        Mediano.Soltar -> Detacher_2.Execute
        Mediano.Soltar -> Detacher_3.Execute
        Mediano.Soltar -> Detacher_4.Execute
        Mediano.Soltar -> Detacher_5.Execute
        Mediano.Soltar -> Detacher_6.Execute
        Mediano.Soltar -> Detacher_7.Execute
        Mediano.Soltar -> Detacher_8.Execute
        Mediano.Coger -> Attacher_18.Execute
        Mediano.Coger -> Attacher_19.Execute
        Mediano.Soltar -> Detacher_9.Execute
        Mediano.Soltar -> Detacher_10.Execute
        Source_4.Executed -> Queue_11.Enqueue
        Source_3.Executed -> Queue_10.Enqueue
        Source_2.Executed -> Queue.DeleteAll
        Detacher.Executed -> Queue_2.DeleteAll
        Detacher_9.Executed -> Queue_10.DeleteAll
        Detacher_10.Executed -> Queue_11.DeleteAll
        Detacher_4.Executed -> Queue_5.DeleteAll
        Detacher_5.Executed -> Queue_6.DeleteAll
        Detacher_6.Executed -> Queue_7.DeleteAll
        Detacher_7.Executed -> Queue_8.DeleteAll
        Detacher_8.Executed -> Queue_9.DeleteAll
        Source_9.Executed -> Mediano.Recoger_med
        Random_2.Executed -> Timer.Interval
        Mediano.Start -> Random_2.Execute
        Source.Copy => Queue.Front
        Queue.Front => LinearMover.Object
        LinearMover.Object => Sink.Object
        Counter.Count => Comparer.ValueA
        Counter.Count => Comparer_2.ValueA
        Counter.Count => Comparer_3.ValueA
        Counter.Count => Comparer_4.ValueA
        Counter.Count => Comparer_5.ValueA
        Counter.Count => Comparer_6.ValueA
        Counter.Count => Comparer_7.ValueA
        Counter.Count => Comparer_8.ValueA
        Counter.Count => ?.ValueA
        Queue_2.Front => Attacher.Child
        Queue_3.Front => Attacher.Child
        Queue_4.Front => Attacher.Child
        Queue_5.Front => Attacher.Child
        Queue_6.Front => Attacher.Child
        Queue_7.Front => Attacher.Child
        Queue_8.Front => Attacher.Child
        Queue_9.Front => Attacher.Child
        Attacher.Child => Detacher.Child
        Source_2.Copy => Queue_2.Front
        Source_3.Copy => Queue_3.Front
        Source_4.Copy => Queue_4.Front
        Source_5.Copy => Queue_5.Front
        Source_6.Copy => Queue_6.Front
        Source_7.Copy => Queue_7.Front
        Source_8.Copy => Queue_8.Front
        Source_9.Copy => Queue_9.Front
        Queue_2.Front => Attacher_3.Child
        Attacher_1.Child => Detacher.Child
        Queue_4.Front => Attacher_5.Parent
        Queue_5.Front => Attacher_5.Child
        Queue_6.Front => Attacher_6.Parent
        Queue_7.Front => Attacher_6.Child
        Queue_8.Front => Attacher_7.Parent
        Queue_9.Front => Attacher_7.Child
        Queue_3.Front => Attacher_2.Child
        Queue_4.Front => Attacher_3.Child
        Queue_5.Front => Attacher_4.Child
        Queue_6.Front => Attacher_5.Child
        Queue_7.Front => Attacher_6.Child
        Queue_8.Front => Attacher_7.Child
        Queue_9.Front => Attacher_8.Child
        Attacher_2.Child => Detacher_2.Child
        Attacher_3.Child => Detacher_3.Child
        Attacher_4.Child => Detacher_4.Child
        Attacher_5.Child => Detacher_5.Child
        Attacher_6.Child => Detacher_6.Child
        Attacher_7.Child => Detacher_7.Child
        Attacher_8.Child => Detacher_8.Child
        Queue_2.Front => Attacher_1.Child
        Queue_3.Front => Attacher_18.Child
        Queue_4.Front => Attacher_19.Child
        Attacher_18.Child => Detacher_2.Child
        Attacher_19.Child => Detacher_3.Child
        Source_4.Copy => Queue_11.Front
        Source_3.Copy => Queue_10.Front
        Queue_10.Front => Attacher_18.Child
        Queue_11.Front => Attacher_19.Child
        Attacher_18.Child => Detacher_9.Child
        Attacher_19.Child => Detacher_10.Child
    - LinearMover [smart component, from Components\LinearMover.rslib]
        properties: Object=(none); Direction=[-0.001 0 0]; Speed=1.5; Reference=Global; ReferenceObject=(none)
    - PlaneSensor [smart component, from Components\PlaneSensor.rslib] at (-2318.14, -838.49, 840.87) mm, rotated rx 0 ry -90 rz 0 deg
        properties: Origin=[0 0 0]; Axis1=[0.2 0 0]; Axis2=[0 0.6 0]; SensedPart=(none)
      - _sensorPart_ [part], size 200 x 600 x 0 mm
    - Detacher [smart component, from Components\Detacher.rslib]
        properties: Child=(none); KeepPosition=true
    - Queue [smart component, from Components\Queue.rslib]
        properties: Back=(none); Front=(none); Queue=; NumberOfObjects=0
    - Source [smart component, from Components\Source.rslib]
        properties: Source=Pieza_19; Copy=(none); Parent=(none); Position=[4.6 -0.22 0.775]; Orientation=[0 0 1.5707963267949]; Transient=true; PhysicsBehavior=0
    - Timer [smart component, from Components\Timer.rslib]
        properties: StartTime=0; Interval=4; Repeat=true; CurrentTime=11.448
    - Sink [smart component, from Components\Sink.rslib]
        properties: Object=(none)
    - Source_2 [smart component, from Components\Source.rslib]
        properties: Source=Pieza_19; Copy=(none); Parent=(none); Position=[1.015 0.19 0.7]; Orientation=[0 0 1.5707963267949]; Transient=false; PhysicsBehavior=0
    - Source_3 [smart component, from Components\Source.rslib]
        properties: Source=Pieza_19; Copy=(none); Parent=(none); Position=[1.345 0.19 0.7]; Orientation=[0 0 1.5707963267949]; Transient=false; PhysicsBehavior=0
    - Source_4 [smart component, from Components\Source.rslib]
        properties: Source=Pieza_19; Copy=(none); Parent=(none); Position=[1.675 0.19 0.7]; Orientation=[0 0 1.5707963267949]; Transient=false; PhysicsBehavior=0
    - Queue_2 [smart component, from Components\Queue.rslib]
        properties: Back=(none); Front=(none); Queue=; NumberOfObjects=0
    - Counter [smart component, from Components\Counter.rslib]
        properties: Count=0
    - LogicGate [smart component, from Components\LogicGate.rslib]
        properties: Operator=AND; Delay=0
    - Comparer [smart component, from Components\Comparer.rslib]
        properties: ValueA=0; Operator===; ValueB=1
    - Comparer_2 [smart component, from Components\Comparer.rslib]
        properties: ValueA=0; Operator===; ValueB=2
    - Comparer_3 [smart component, from Components\Comparer.rslib]
        properties: ValueA=0; Operator===; ValueB=3
    - Comparer_4 [smart component, from Components\Comparer.rslib]
        properties: ValueA=0; Operator===; ValueB=4
    - Comparer_5 [smart component, from Components\Comparer.rslib]
        properties: ValueA=0; Operator===; ValueB=5
    - Comparer_6 [smart component, from Components\Comparer.rslib]
        properties: ValueA=0; Operator===; ValueB=6
    - Comparer_7 [smart component, from Components\Comparer.rslib]
        properties: ValueA=0; Operator===; ValueB=7
    - LogicGate_2 [smart component, from Components\LogicGate.rslib]
        properties: Operator=AND; Delay=0
    - LogicGate_3 [smart component, from Components\LogicGate.rslib]
        properties: Operator=AND; Delay=0
    - LogicGate_4 [smart component, from Components\LogicGate.rslib]
        properties: Operator=AND; Delay=0
    - LogicGate_5 [smart component, from Components\LogicGate.rslib]
        properties: Operator=AND; Delay=0
    - LogicGate_6 [smart component, from Components\LogicGate.rslib]
        properties: Operator=AND; Delay=0
    - LogicGate_7 [smart component, from Components\LogicGate.rslib]
        properties: Operator=AND; Delay=0
    - Queue_5 [smart component, from Components\Queue.rslib]
        properties: Back=(none); Front=(none); Queue=; NumberOfObjects=0
    - Queue_6 [smart component, from Components\Queue.rslib]
        properties: Back=(none); Front=(none); Queue=; NumberOfObjects=0
    - Queue_7 [smart component, from Components\Queue.rslib]
        properties: Back=(none); Front=(none); Queue=; NumberOfObjects=0
    - Queue_8 [smart component, from Components\Queue.rslib]
        properties: Back=(none); Front=(none); Queue=; NumberOfObjects=0
    - Source_5 [smart component, from Components\Source.rslib]
        properties: Source=Pieza_19; Copy=(none); Parent=(none); Position=[0.69 -0.14 0.7]; Orientation=[0 0 0]; Transient=false; PhysicsBehavior=0
    - Source_6 [smart component, from Components\Source.rslib]
        properties: Source=Pieza_19; Copy=(none); Parent=(none); Position=[1.255 -0.14 0.7]; Orientation=[0 0 0]; Transient=false; PhysicsBehavior=0
    - Source_7 [smart component, from Components\Source.rslib]
        properties: Source=Pieza_19; Copy=(none); Parent=(none); Position=[1.015 -0.57 0.7]; Orientation=[0 0 1.5707963267949]; Transient=false; PhysicsBehavior=0
    - Source_8 [smart component, from Components\Source.rslib]
        properties: Source=Pieza_19; Copy=(none); Parent=(none); Position=[1.345 -0.57 0.7]; Orientation=[0 0 1.5707963267949]; Transient=false; PhysicsBehavior=0
    - Comparer_8 [smart component, from Components\Comparer.rslib]
        properties: ValueA=0; Operator=>=; ValueB=8
    - Source_9 [smart component, from Components\Source.rslib]
        properties: Source=Pieza_19; Copy=(none); Parent=(none); Position=[1.675 -0.57 0.7]; Orientation=[0 0 1.5707963267949]; Transient=false; PhysicsBehavior=0
    - Queue_9 [smart component, from Components\Queue.rslib]
        properties: Back=(none); Front=(none); Queue=; NumberOfObjects=0
    - LogicGate_8 [smart component, from Components\LogicGate.rslib]
        properties: Operator=AND; Delay=0
    - Attacher_1 [smart component, from Components\Attacher.rslib]
        properties: Parent=Mi_mecanismo; Flange=0; Child=(none); Mount=false; Offset=[0 0 0]; Orientation=[0 0 0]
    - Attacher_4 [smart component, from Components\Attacher.rslib]
        properties: Parent=Mi_mecanismo; Flange=0; Child=(none); Mount=false; Offset=[0 0 0]; Orientation=[0 0 0]
    - Attacher_5 [smart component, from Components\Attacher.rslib]
        properties: Parent=Mi_mecanismo; Flange=0; Child=(none); Mount=false; Offset=[0 0 0]; Orientation=[0 0 0]
    - Attacher_6 [smart component, from Components\Attacher.rslib]
        properties: Parent=Mi_mecanismo; Flange=0; Child=(none); Mount=false; Offset=[0 0 0]; Orientation=[0 0 0]
    - Attacher_7 [smart component, from Components\Attacher.rslib]
        properties: Parent=Mi_mecanismo; Flange=0; Child=(none); Mount=false; Offset=[0 0 0]; Orientation=[0 0 0]
    - Attacher_8 [smart component, from Components\Attacher.rslib]
        properties: Parent=Mi_mecanismo; Flange=0; Child=(none); Mount=false; Offset=[0 0 0]; Orientation=[0 0 0]
    - Detacher_4 [smart component, from Components\Detacher.rslib]
        properties: Child=(none); KeepPosition=true
    - Detacher_5 [smart component, from Components\Detacher.rslib]
        properties: Child=(none); KeepPosition=true
    - Detacher_6 [smart component, from Components\Detacher.rslib]
        properties: Child=(none); KeepPosition=true
    - Detacher_7 [smart component, from Components\Detacher.rslib]
        properties: Child=(none); KeepPosition=true
    - Detacher_8 [smart component, from Components\Detacher.rslib]
        properties: Child=(none); KeepPosition=true
    - Attacher_18 [smart component, from Components\Attacher.rslib]
        properties: Parent=Mi_mecanismo; Flange=0; Child=(none); Mount=false; Offset=[0 0 0]; Orientation=[0 0 0]
    - Attacher_19 [smart component, from Components\Attacher.rslib]
        properties: Parent=Mi_mecanismo; Flange=0; Child=(none); Mount=false; Offset=[0 0 0]; Orientation=[0 0 0]
    - Detacher_9 [smart component, from Components\Detacher.rslib]
        properties: Child=(none); KeepPosition=true
    - Detacher_10 [smart component, from Components\Detacher.rslib]
        properties: Child=(none); KeepPosition=true
    - Queue_10 [smart component, from Components\Queue.rslib]
        properties: Back=(none); Front=(none); Queue=; NumberOfObjects=0
    - Queue_11 [smart component, from Components\Queue.rslib]
        properties: Back=(none); Front=(none); Queue=; NumberOfObjects=0
Attachment: Mi_mecanismo is attached to IRB660_180_315__01 / Link6
Attachment: PlaneSensor is attached to 1200_4800_h2_2
EventTableEntry 2667: Group=, Trigger=Agarrar 2668, Actions=[EventTableActionMechanicalPose 2669], Comment=, ActivationMode=2, Cyclic=false
EventTableTriggerIO 2668: IOValue=[1], IRC5Controller=? -1, Operator=0, SignalSource=IRB660_180_315 1167
EventTableActionMechanicalPose 2669: VirtualSignal=, Mechanism=Mi_mecanismo 2358, ToPoseName=Pose final, VirtualSignalValue=[1]
EventTableEntry 2670: Group=, Trigger=Agarrar 2671, Actions=[EventTableActionMechanicalPose 2672], Comment=, ActivationMode=2, Cyclic=false
EventTableTriggerIO 2671: IOValue=[0], IRC5Controller=? -1, Operator=0, SignalSource=IRB660_180_315 1167
EventTableActionMechanicalPose 2672: VirtualSignal=, Mechanism=Mi_mecanismo 2358, ToPoseName=HomePosition, VirtualSignalValue=[1]
EventTableTriggerIO 2976: IOValue=[1], IRC5Controller=? -1, Operator=0, SignalSource=IRB660_180_315 1167
EventTableTriggerIO 2977: IOValue=[1], IRC5Controller=? -1, Operator=0, SignalSource=IRB660_180_315 1167
EventTableTriggerIO 2978: IOValue=[0], IRC5Controller=? -1, Operator=0, SignalSource=IRB660_180_315 1167
EventTableTriggerIO 2979: IOValue=[0], IRC5Controller=? -1, Operator=0, SignalSource=IRB660_180_315 1167
EventTableTriggerIO 3572: IOValue=[1], IRC5Controller=? -1, Operator=0, SignalSource=IRB660_180_315 1167
EventTableTriggerIO 3573: IOValue=[1], IRC5Controller=? -1, Operator=0, SignalSource=IRB660_180_315 1167
EventTableTriggerIO 3574: IOValue=[1], IRC5Controller=? -1, Operator=0, SignalSource=IRB660_180_315 1167
EventTableTriggerIO 3575: IOValue=[1], IRC5Controller=? -1, Operator=0, SignalSource=IRB660_180_315 1167
EventTableTriggerIO 3576: IOValue=[1], IRC5Controller=? -1, Operator=0, SignalSource=IRB660_180_315 1167
EventTableTriggerIO 3577: IOValue=[1], IRC5Controller=? -1, Operator=0, SignalSource=IRB660_180_315 1167
EventTableTriggerIO 3578: IOValue=[1], IRC5Controller=? -1, Operator=0, SignalSource=IRB660_180_315 1167
EventTableTriggerIO 3579: IOValue=[1], IRC5Controller=? -1, Operator=0, SignalSource=IRB660_180_315 1167
EventTableTriggerIO 3580: IOValue=[1], IRC5Controller=? -1, Operator=0, SignalSource=IRB660_180_315 1167
EventTableTriggerIO 3581: IOValue=[1], IRC5Controller=? -1, Operator=0, SignalSource=IRB660_180_315 1167
EventTableTriggerIO 3582: IOValue=[0], IRC5Controller=? -1, Operator=0, SignalSource=IRB660_180_315 1167
EventTableTriggerIO 3583: IOValue=[0], IRC5Controller=? -1, Operator=0, SignalSource=IRB660_180_315 1167
EventTableTriggerIO 3584: IOValue=[0], IRC5Controller=? -1, Operator=0, SignalSource=IRB660_180_315 1167
EventTableTriggerIO 3585: IOValue=[0], IRC5Controller=? -1, Operator=0, SignalSource=IRB660_180_315 1167
EventTableTriggerIO 3586: IOValue=[0], IRC5Controller=? -1, Operator=0, SignalSource=IRB660_180_315 1167
EventTableTriggerIO 3587: IOValue=[0], IRC5Controller=? -1, Operator=0, SignalSource=IRB660_180_315 1167
EventTableTriggerIO 3588: IOValue=[0], IRC5Controller=? -1, Operator=0, SignalSource=IRB660_180_315 1167
EventTableTriggerIO 3589: IOValue=[0], IRC5Controller=? -1, Operator=0, SignalSource=IRB660_180_315 1167
EventTableTriggerIO 3590: IOValue=[0], IRC5Controller=? -1, Operator=0, SignalSource=IRB660_180_315 1167
EventTableTriggerIO 3591: IOValue=[0], IRC5Controller=? -1, Operator=0, SignalSource=IRB660_180_315 1167
Station logic (signal -> signal, property => property):
  IRB660_180_315.StartRob -> Pequeño.Start
  IRB660_180_315.CintaRob -> Pequeño.Cinta
  IRB660_180_315.CogerRob -> Pequeño.Coger
  IRB660_180_315.SoltarRob -> Pequeño.Soltar
  Pequeño.Sensor1 -> IRB660_180_315.Sensor1Rob
  Pequeño.Recoger_peq -> IRB660_180_315.Recoger_peq_rob
  IRB660_180_315.Start_med -> Mediano.Start
  IRB660_180_315.Cinta_med -> Mediano.Cinta
  IRB660_180_315.Coger_med -> Mediano.Coger
  IRB660_180_315.Soltar_med -> Mediano.Soltar
  Mediano.Sensor1 -> IRB660_180_315.Sensor1_med
  Mediano.Recoger_med -> IRB660_180_315.Recoger_med
  IRB660_180_315.Start_gra -> Grande.Start
  IRB660_180_315.Cinta_gra -> Grande.Cinta
  IRB660_180_315.Coger_gra -> Grande.Coger
  IRB660_180_315.Soltar_gra -> Grande.Soltar
  Grande.Sensor1 -> IRB660_180_315.Sensor1_gra
  Grande.Recoger_peq -> IRB660_180_315.Recocger_gra
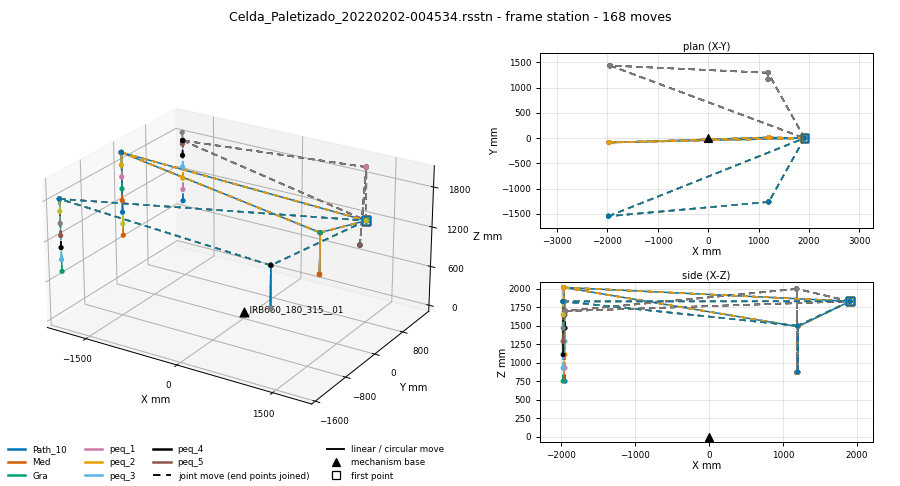
[picture p0: tool path of Celda_Paletizado_20220202-004534.rsstn in frame station, 168 of 168 moves have a stored position in this frame; points joined in program order, loops and branches not executed]
Targets, tools, work objects and paths stored in the station, written as RAPID:
! task T_ROB1
MODULE CalibData
  TASK PERS wobjdata pequeño:=[FALSE,TRUE,"",[[0,0,0],[1,0,0,0]],[[0,0,0],[1,0,0,0]]];
  TASK PERS wobjdata Mediano:=[FALSE,TRUE,"",[[0,0,0],[1,0,0,0]],[[0,0,0],[1,0,0,0]]];
  TASK PERS wobjdata Grande:=[FALSE,TRUE,"",[[0,0,0],[1,0,0,0]],[[0,0,0],[1,0,0,0]]];
  PERS tooldata Servo:=[TRUE,[[0,0,114.2],[1,0,0,0]],[0.215,[8.7,12.3,49.2],[1,0,0,0],0.00021,0.00024,0.00009]];
  PERS tooldata Gripper:=[TRUE,[[0,-0.226,3866.059],[1,0,0,0]],[60,[0,0,200],[1,0,0,0],0,0,0]];
  PERS tooldata Mi_mecanismo_1:=[TRUE,[[0,0,260],[1,0,0,0]],[60,[0,0,-280],[1,0,0,0],0,0,0]];
  TASK PERS wobjdata Workobject_1:=[FALSE,TRUE,"",[[0,0,0],[1,0,0,0]],[[0,0,0],[1,0,0,0]]];
  TASK PERS wobjdata Workobject_2:=[FALSE,TRUE,"",[[0,0,0],[1,0,0,0]],[[0,0,0],[1,0,0,0]]];
ENDMODULE

! task T_ROB1
MODULE Module1
  CONST robtarget Home:=[[1909.999941719,0,1832.999945473],[0,0,1,0],[0,0,0,0],[9E+09,9E+09,9E+09,9E+09,9E+09,9E+09]];
  CONST robtarget Target_10:=[[1189.01,1165.635,870],[0,0,1,0],[0,0,0,0],[9E+09,9E+09,9E+09,9E+09,9E+09,9E+09]];
  CONST robtarget Target_20:=[[1189.01,1295.635,2000],[0,0,1,0],[0,0,0,0],[9E+09,9E+09,9E+09,9E+09,9E+09,9E+09]];
  CONST robtarget Target_30:=[[-1945,1440,1700],[0,0,1,0],[0,0,0,0],[9E+09,9E+09,9E+09,9E+09,9E+09,9E+09]];
  CONST robtarget Target_40:=[[-1945,1430,750],[0,0,1,0],[0,0,0,0],[9E+09,9E+09,9E+09,9E+09,9E+09,9E+09]];
  CONST robtarget Target_50:=[[1203.573,14.679,870],[0,0,1,0],[0,0,0,0],[9E+09,9E+09,9E+09,9E+09,9E+09,9E+09]];
  CONST robtarget Target_60:=[[1203.573,14.679,1490.240493886],[0,0,1,0],[0,0,0,0],[9E+09,9E+09,9E+09,9E+09,9E+09,9E+09]];
  CONST robtarget Target_70:=[[-1965.701,-87.059,753.354],[0,0,1,0],[0,0,0,0],[9E+09,9E+09,9E+09,9E+09,9E+09,9E+09]];
  CONST robtarget Target_80:=[[-1965.701,-87.059,2020],[0,0,1,0],[0,0,0,0],[9E+09,9E+09,9E+09,9E+09,9E+09,9E+09]];
  CONST robtarget Target_90:=[[1202.605,-1263.746,876],[0,0,1,0],[0,0,0,0],[9E+09,9E+09,9E+09,9E+09,9E+09,9E+09]];
  CONST robtarget Target_100:=[[1202.605,-1263.746,1500],[0,0,1,0],[0,0,0,0],[9E+09,9E+09,9E+09,9E+09,9E+09,9E+09]];
  CONST robtarget Target_110:=[[-1975,-1547.039,752.357],[0,0,1,0],[0,0,0,0],[9E+09,9E+09,9E+09,9E+09,9E+09,9E+09]];
  CONST robtarget Target_120:=[[-1975,-1547.039,1831],[0,0,1,0],[0,0,0,0],[9E+09,9E+09,9E+09,9E+09,9E+09,9E+09]];
  CONST robtarget Target_130:=[[-1975,-1550,930],[0,0,1,0],[0,0,0,0],[9E+09,9E+09,9E+09,9E+09,9E+09,9E+09]];
  CONST robtarget Target_140:=[[-1975,-1550,1110],[0,0,1,0],[0,0,0,0],[9E+09,9E+09,9E+09,9E+09,9E+09,9E+09]];
  CONST robtarget Target_150:=[[-1975,-1550,1290],[0,0,1,0],[0,0,0,0],[9E+09,9E+09,9E+09,9E+09,9E+09,9E+09]];
  CONST robtarget Target_160:=[[-1975,-1550,1470],[0,0,1,0],[0,0,0,0],[9E+09,9E+09,9E+09,9E+09,9E+09,9E+09]];
  CONST robtarget Target_170:=[[-1975,-1550,1650],[0,0,1,0],[0,0,0,0],[9E+09,9E+09,9E+09,9E+09,9E+09,9E+09]];
  CONST robtarget Target_180:=[[-1975,-1550,1830],[0,0,1,0],[0,0,0,0],[9E+09,9E+09,9E+09,9E+09,9E+09,9E+09]];
  CONST robtarget Target_190:=[[-1967,-90,750],[0,0,1,0],[0,0,0,0],[9E+09,9E+09,9E+09,9E+09,9E+09,9E+09]];
  CONST robtarget Target_200:=[[-1967,-90,930],[0,0,1,0],[0,0,0,0],[9E+09,9E+09,9E+09,9E+09,9E+09,9E+09]];
  CONST robtarget Target_210:=[[-1967,-90,1110],[0,0,1,0],[0,0,0,0],[9E+09,9E+09,9E+09,9E+09,9E+09,9E+09]];
  CONST robtarget Target_220:=[[-1967,-90,1290],[0,0,1,0],[0,0,0,0],[9E+09,9E+09,9E+09,9E+09,9E+09,9E+09]];
  CONST robtarget Target_230:=[[-1967,-90,1470],[0,0,1,0],[0,0,0,0],[9E+09,9E+09,9E+09,9E+09,9E+09,9E+09]];
  CONST robtarget Target_240:=[[-1967,-90,1650],[0,0,1,0],[0,0,0,0],[9E+09,9E+09,9E+09,9E+09,9E+09,9E+09]];
  CONST robtarget Target_250:=[[-1967,-90,1830],[0,0,1,0],[0,0,0,0],[9E+09,9E+09,9E+09,9E+09,9E+09,9E+09]];
  CONST robtarget Target_260:=[[-1945,1430,750],[0,0,1,0],[0,0,0,0],[9E+09,9E+09,9E+09,9E+09,9E+09,9E+09]];
  CONST robtarget Target_270:=[[-1945,1430,930],[0,0,1,0],[0,0,0,0],[9E+09,9E+09,9E+09,9E+09,9E+09,9E+09]];
  CONST robtarget Target_280:=[[-1945,1430,1110],[0,0,1,0],[0,0,0,0],[9E+09,9E+09,9E+09,9E+09,9E+09,9E+09]];
  CONST robtarget Target_290:=[[-1945,1430,1290],[0,0,1,0],[0,0,0,0],[9E+09,9E+09,9E+09,9E+09,9E+09,9E+09]];
  CONST robtarget Target_300:=[[-1945,1430,1470],[0,0,1,0],[0,0,0,0],[9E+09,9E+09,9E+09,9E+09,9E+09,9E+09]];
  CONST robtarget Target_310:=[[-1945,1430,1650],[0,0,1,0],[0,0,0,0],[9E+09,9E+09,9E+09,9E+09,9E+09,9E+09]];
  CONST robtarget Target_320:=[[-1945,1430,1830],[0,0,1,0],[0,0,0,0],[9E+09,9E+09,9E+09,9E+09,9E+09,9E+09]];
  PROC Path_10()
    MoveJ Home,v7000,fine,Mi_mecanismo_1\WObj:=wobj0;
    MoveJ Target_20,v7000,fine,Mi_mecanismo_1\WObj:=wobj0;
    SetDO Agarrar,1;
    MoveJ Target_10,v7000,fine,Mi_mecanismo_1\WObj:=wobj0;
    SetDO CogerRob,1;
    SetDO Agarrar,0;
    SetDO CintaRob,1;
    MoveJ Target_20,v7000,fine,Mi_mecanismo_1\WObj:=wobj0;
    MoveJ Target_30,v7000,fine,Mi_mecanismo_1\WObj:=wobj0;
    MoveJ Target_40,v7000,fine,Mi_mecanismo_1\WObj:=wobj0;
    SetDO CogerRob,0;
    SetDO SoltarRob,1;
    SetDO Agarrar,1;
    MoveJ Target_30,v7000,fine,Mi_mecanismo_1\WObj:=wobj0;
    SetDO Agarrar,0;
    MoveJ Home,v7000,fine,Mi_mecanismo_1\WObj:=wobj0;
    SetDO SoltarRob,0;
  ENDPROC
  PROC main()
    SetDO CogerRob,0;
    SetDO SoltarRob,0;
    SetDO StartRob,1;
    SetDO CintaRob,1;
    SetDO Coger_med,0;
    SetDO Soltar_med,0;
    SetDO Start_med,1;
    SetDO Cinta_med,1;
    SetDO Coger_gra,0;
    SetDO Soltar_gra,0;
    SetDO Start_gra,1;
    SetDO Cinta_gra,1;
    Path_10;
    peq_1;
    peq_2;
    peq_3;
    peq_4;
    peq_5;
    peq_6;
    Med;
    med_1;
    med_2;
    med_3;
    med_4;
    med_5;
    med_6;
    Gra;
    gra_1;
    gra_2;
    gra_3;
    gra_4;
    gra_5;
    gra_6;
  ENDPROC
  PROC Med()
    MoveJ Home,v7000,fine,Mi_mecanismo_1\WObj:=wobj0;
    MoveJ Target_60,v7000,fine,Mi_mecanismo_1\WObj:=Workobject_1;
    SetDO Agarrar,1;
    MoveJ Target_50,v7000,fine,Mi_mecanismo_1\WObj:=Workobject_1;
    SetDO Coger_med,1;
    SetDO Agarrar,0;
    SetDO Cinta_med,1;
    MoveJ Target_60,v7000,fine,Mi_mecanismo_1\WObj:=Workobject_1;
    MoveJ Target_80,v7000,fine,Mi_mecanismo_1\WObj:=Workobject_1;
    MoveJ Target_70,v7000,fine,Mi_mecanismo_1\WObj:=Workobject_1;
    SetDO Coger_med,0;
    SetDO Soltar_med,1;
    SetDO Agarrar,1;
    MoveJ Target_80,v7000,fine,Mi_mecanismo_1\WObj:=Workobject_1;
    SetDO Agarrar,0;
    MoveJ Home,v7000,fine,Mi_mecanismo_1\WObj:=wobj0;
    SetDO Soltar_med,0;
  ENDPROC
  PROC Gra()
    MoveJ Home,v7000,fine,Mi_mecanismo_1\WObj:=wobj0;
    MoveJ Target_100,v7000,fine,Mi_mecanismo_1\WObj:=Workobject_2;
    SetDO Agarrar,1;
    MoveJ Target_90,v7000,fine,Mi_mecanismo_1\WObj:=Workobject_2;
    SetDO Coger_gra,1;
    SetDO Cinta_gra,1;
    SetDO Agarrar,0;
    MoveJ Target_100,v7000,fine,Mi_mecanismo_1\WObj:=Workobject_2;
    MoveJ Target_120,v7000,fine,Mi_mecanismo_1\WObj:=Workobject_2;
    MoveJ Target_110,v7000,fine,Mi_mecanismo_1\WObj:=Workobject_2;
    SetDO Coger_gra,0;
    SetDO Soltar_gra,1;
    SetDO Agarrar,1;
    MoveJ Target_120,v7000,fine,Mi_mecanismo_1\WObj:=Workobject_2;
    SetDO Agarrar,0;
    MoveJ Home,v7000,fine,Mi_mecanismo_1\WObj:=wobj0;
    SetDO Soltar_gra,0;
  ENDPROC
  PROC peq_1()
    MoveJ Home,v7000,fine,Mi_mecanismo_1\WObj:=wobj0;
    MoveJ Target_20,v7000,fine,Mi_mecanismo_1\WObj:=wobj0;
    SetDO Agarrar,1;
    MoveJ Target_10,v7000,fine,Mi_mecanismo_1\WObj:=wobj0;
    SetDO CogerRob,1;
    SetDO Agarrar,0;
    SetDO CintaRob,1;
    MoveJ Target_20,v7000,fine,Mi_mecanismo_1\WObj:=wobj0;
    MoveJ Target_30,v7000,fine,Mi_mecanismo_1\WObj:=wobj0;
    MoveJ Target_270,v7000,fine,Mi_mecanismo_1\WObj:=wobj0;
    SetDO CogerRob,0;
    SetDO SoltarRob,1;
    SetDO Agarrar,1;
    MoveJ Target_30,v7000,fine,Mi_mecanismo_1\WObj:=wobj0;
    SetDO Agarrar,0;
    MoveJ Home,v7000,fine,Mi_mecanismo_1\WObj:=wobj0;
    SetDO SoltarRob,0;
  ENDPROC
  PROC peq_2()
    MoveJ Home,v7000,fine,Mi_mecanismo_1\WObj:=wobj0;
    MoveJ Target_20,v7000,fine,Mi_mecanismo_1\WObj:=wobj0;
    SetDO Agarrar,1;
    MoveJ Target_10,v7000,fine,Mi_mecanismo_1\WObj:=wobj0;
    SetDO CogerRob,1;
    SetDO Agarrar,0;
    SetDO CintaRob,1;
    MoveJ Target_20,v7000,fine,Mi_mecanismo_1\WObj:=wobj0;
    MoveJ Target_30,v7000,fine,Mi_mecanismo_1\WObj:=wobj0;
    MoveJ Target_280,v7000,fine,Mi_mecanismo_1\WObj:=wobj0;
    SetDO CogerRob,0;
    SetDO SoltarRob,1;
    SetDO Agarrar,1;
    MoveJ Target_30,v7000,fine,Mi_mecanismo_1\WObj:=wobj0;
    SetDO Agarrar,0;
    MoveJ Home,v7000,fine,Mi_mecanismo_1\WObj:=wobj0;
    SetDO SoltarRob,0;
  ENDPROC
  PROC peq_3()
    MoveJ Home,v7000,fine,Mi_mecanismo_1\WObj:=wobj0;
    MoveJ Target_20,v7000,fine,Mi_mecanismo_1\WObj:=wobj0;
    SetDO Agarrar,1;
    MoveJ Target_10,v7000,fine,Mi_mecanismo_1\WObj:=wobj0;
    SetDO CogerRob,1;
    SetDO Agarrar,0;
    SetDO CintaRob,1;
    MoveJ Target_20,v7000,fine,Mi_mecanismo_1\WObj:=wobj0;
    MoveJ Target_30,v7000,fine,Mi_mecanismo_1\WObj:=wobj0;
    MoveJ Target_290,v7000,fine,Mi_mecanismo_1\WObj:=wobj0;
    SetDO CogerRob,0;
    SetDO SoltarRob,1;
    SetDO Agarrar,1;
    MoveJ Target_30,v7000,fine,Mi_mecanismo_1\WObj:=wobj0;
    SetDO Agarrar,0;
    MoveJ Home,v7000,fine,Mi_mecanismo_1\WObj:=wobj0;
    SetDO SoltarRob,0;
  ENDPROC
  PROC peq_4()
    MoveJ Home,v7000,fine,Mi_mecanismo_1\WObj:=wobj0;
    MoveJ Target_20,v7000,fine,Mi_mecanismo_1\WObj:=wobj0;
    SetDO Agarrar,1;
    MoveJ Target_10,v7000,fine,Mi_mecanismo_1\WObj:=wobj0;
    SetDO CogerRob,1;
    SetDO Agarrar,0;
    SetDO CintaRob,1;
    MoveJ Target_20,v7000,fine,Mi_mecanismo_1\WObj:=wobj0;
    MoveJ Target_30,v7000,fine,Mi_mecanismo_1\WObj:=wobj0;
    MoveJ Target_300,v7000,fine,Mi_mecanismo_1\WObj:=wobj0;
    SetDO CogerRob,0;
    SetDO SoltarRob,1;
    SetDO Agarrar,1;
    MoveJ Target_30,v7000,fine,Mi_mecanismo_1\WObj:=wobj0;
    SetDO Agarrar,0;
    MoveJ Home,v7000,fine,Mi_mecanismo_1\WObj:=wobj0;
    SetDO SoltarRob,0;
  ENDPROC
  PROC peq_5()
    MoveJ Home,v7000,fine,Mi_mecanismo_1\WObj:=wobj0;
    MoveJ Target_20,v7000,fine,Mi_mecanismo_1\WObj:=wobj0;
    SetDO Agarrar,1;
    MoveJ Target_10,v7000,fine,Mi_mecanismo_1\WObj:=wobj0;
    SetDO CogerRob,1;
    SetDO Agarrar,0;
    SetDO CintaRob,1;
    MoveJ Target_20,v7000,fine,Mi_mecanismo_1\WObj:=wobj0;
    MoveJ Target_30,v7000,fine,Mi_mecanismo_1\WObj:=wobj0;
    MoveJ Target_310,v7000,fine,Mi_mecanismo_1\WObj:=wobj0;
    SetDO CogerRob,0;
    SetDO SoltarRob,1;
    SetDO Agarrar,1;
    MoveJ Target_30,v7000,fine,Mi_mecanismo_1\WObj:=wobj0;
    SetDO Agarrar,0;
    MoveJ Home,v7000,fine,Mi_mecanismo_1\WObj:=wobj0;
    SetDO SoltarRob,0;
  ENDPROC
  PROC peq_6()
    MoveJ Home,v7000,fine,Mi_mecanismo_1\WObj:=wobj0;
    MoveJ Target_20,v7000,fine,Mi_mecanismo_1\WObj:=wobj0;
    SetDO Agarrar,1;
    MoveJ Target_10,v7000,fine,Mi_mecanismo_1\WObj:=wobj0;
    SetDO CogerRob,1;
    SetDO Agarrar,0;
    SetDO CintaRob,1;
    MoveJ Target_20,v7000,fine,Mi_mecanismo_1\WObj:=wobj0;
    MoveJ Target_30,v7000,fine,Mi_mecanismo_1\WObj:=wobj0;
    MoveJ Target_320,v7000,fine,Mi_mecanismo_1\WObj:=wobj0;
    SetDO CogerRob,0;
    SetDO SoltarRob,1;
    SetDO Agarrar,1;
    MoveJ Target_30,v7000,fine,Mi_mecanismo_1\WObj:=wobj0;
    SetDO Agarrar,0;
    MoveJ Home,v7000,fine,Mi_mecanismo_1\WObj:=wobj0;
    SetDO SoltarRob,0;
  ENDPROC
  PROC med_1()
    MoveJ Home,v7000,fine,Mi_mecanismo_1\WObj:=wobj0;
    MoveJ Target_60,v7000,fine,Mi_mecanismo_1\WObj:=Workobject_1;
    SetDO Agarrar,1;
    MoveJ Target_50,v7000,fine,Mi_mecanismo_1\WObj:=Workobject_1;
    SetDO Coger_med,1;
    SetDO Agarrar,0;
    SetDO Cinta_med,1;
    MoveJ Target_60,v7000,fine,Mi_mecanismo_1\WObj:=Workobject_1;
    MoveJ Target_80,v7000,fine,Mi_mecanismo_1\WObj:=Workobject_1;
    MoveJ Target_200,v7000,fine,Mi_mecanismo_1\WObj:=Workobject_1;
    SetDO Coger_med,0;
    SetDO Soltar_med,1;
    SetDO Agarrar,1;
    MoveJ Target_80,v7000,fine,Mi_mecanismo_1\WObj:=Workobject_1;
    SetDO Agarrar,0;
    MoveJ Home,v7000,fine,Mi_mecanismo_1\WObj:=wobj0;
    SetDO Soltar_med,0;
  ENDPROC
  PROC med_2()
    MoveL Home,v7000,fine,Mi_mecanismo_1\WObj:=wobj0;
    MoveL Target_60,v7000,fine,Mi_mecanismo_1\WObj:=Workobject_1;
    SetDO Agarrar,1;
    MoveL Target_50,v7000,fine,Mi_mecanismo_1\WObj:=Workobject_1;
    SetDO Coger_med,1;
    SetDO Agarrar,0;
    SetDO Cinta_med,1;
    MoveL Target_60,v7000,fine,Mi_mecanismo_1\WObj:=Workobject_1;
    MoveL Target_80,v7000,fine,Mi_mecanismo_1\WObj:=Workobject_1;
    MoveL Target_210,v1000,z100,Mi_mecanismo_1\WObj:=Workobject_1;
    SetDO Coger_med,0;
    SetDO Soltar_med,1;
    SetDO Agarrar,1;
    MoveL Target_80,v7000,fine,Mi_mecanismo_1\WObj:=Workobject_1;
    SetDO Agarrar,0;
    MoveL Home,v7000,fine,Mi_mecanismo_1\WObj:=wobj0;
    SetDO Soltar_med,0;
  ENDPROC
  PROC med_3()
    MoveJ Home,v7000,fine,Mi_mecanismo_1\WObj:=wobj0;
    MoveJ Target_60,v7000,fine,Mi_mecanismo_1\WObj:=Workobject_1;
    SetDO Agarrar,1;
    MoveJ Target_50,v7000,fine,Mi_mecanismo_1\WObj:=Workobject_1;
    SetDO Coger_med,1;
    SetDO Agarrar,0;
    SetDO Cinta_med,1;
    MoveJ Target_60,v7000,fine,Mi_mecanismo_1\WObj:=Workobject_1;
    MoveJ Target_80,v7000,fine,Mi_mecanismo_1\WObj:=Workobject_1;
    MoveJ Target_220,v7000,fine,Mi_mecanismo_1\WObj:=Workobject_1;
    SetDO Coger_med,0;
    SetDO Soltar_med,1;
    SetDO Agarrar,1;
    MoveJ Target_80,v7000,fine,Mi_mecanismo_1\WObj:=Workobject_1;
    SetDO Agarrar,0;
    MoveJ Home,v7000,fine,Mi_mecanismo_1\WObj:=wobj0;
    SetDO Soltar_med,0;
  ENDPROC
  PROC med_4()
    MoveJ Home,v7000,fine,Mi_mecanismo_1\WObj:=wobj0;
    MoveJ Target_60,v7000,fine,Mi_mecanismo_1\WObj:=Workobject_1;
    SetDO Agarrar,1;
    MoveJ Target_50,v7000,fine,Mi_mecanismo_1\WObj:=Workobject_1;
    SetDO Coger_med,1;
    SetDO Agarrar,0;
    SetDO Cinta_med,1;
    MoveJ Target_60,v7000,fine,Mi_mecanismo_1\WObj:=Workobject_1;
    MoveJ Target_80,v7000,fine,Mi_mecanismo_1\WObj:=Workobject_1;
    MoveJ Target_230,v7000,fine,Mi_mecanismo_1\WObj:=Workobject_1;
    SetDO Coger_med,0;
    SetDO Soltar_med,1;
    SetDO Agarrar,1;
    MoveJ Target_80,v7000,fine,Mi_mecanismo_1\WObj:=Workobject_1;
    SetDO Agarrar,0;
    MoveJ Home,v7000,fine,Mi_mecanismo_1\WObj:=wobj0;
    SetDO Soltar_med,0;
  ENDPROC
  PROC med_5()
    MoveJ Home,v7000,fine,Mi_mecanismo_1\WObj:=wobj0;
    MoveJ Target_60,v7000,fine,Mi_mecanismo_1\WObj:=Workobject_1;
    SetDO Agarrar,1;
    MoveJ Target_50,v7000,fine,Mi_mecanismo_1\WObj:=Workobject_1;
    SetDO Coger_med,1;
    SetDO Agarrar,0;
    SetDO Cinta_med,1;
    MoveJ Target_60,v7000,fine,Mi_mecanismo_1\WObj:=Workobject_1;
    MoveJ Target_80,v7000,fine,Mi_mecanismo_1\WObj:=Workobject_1;
    MoveJ Target_240,v7000,fine,Mi_mecanismo_1\WObj:=Workobject_1;
    SetDO Coger_med,0;
    SetDO Soltar_med,1;
    SetDO Agarrar,1;
    MoveJ Target_80,v7000,fine,Mi_mecanismo_1\WObj:=Workobject_1;
    SetDO Agarrar,0;
    MoveJ Home,v7000,fine,Mi_mecanismo_1\WObj:=wobj0;
    SetDO Soltar_med,0;
  ENDPROC
  PROC med_6()
    MoveJ Home,v7000,fine,Mi_mecanismo_1\WObj:=wobj0;
    MoveJ Target_60,v7000,fine,Mi_mecanismo_1\WObj:=Workobject_1;
    SetDO Agarrar,1;
    MoveJ Target_50,v7000,fine,Mi_mecanismo_1\WObj:=Workobject_1;
    SetDO Coger_med,1;
    SetDO Agarrar,0;
    SetDO Cinta_med,1;
    MoveJ Target_60,v7000,fine,Mi_mecanismo_1\WObj:=Workobject_1;
    MoveJ Target_80,v7000,fine,Mi_mecanismo_1\WObj:=Workobject_1;
    MoveJ Target_250,v7000,fine,Mi_mecanismo_1\WObj:=Workobject_1;
    SetDO Coger_med,0;
    SetDO Soltar_med,1;
    SetDO Agarrar,1;
    MoveJ Target_80,v7000,fine,Mi_mecanismo_1\WObj:=Workobject_1;
    SetDO Agarrar,0;
    MoveJ Home,v7000,fine,Mi_mecanismo_1\WObj:=wobj0;
    SetDO Soltar_med,0;
  ENDPROC
  PROC gra_1()
    MoveJ Home,v7000,fine,Mi_mecanismo_1\WObj:=wobj0;
    MoveJ Target_100,v7000,fine,Mi_mecanismo_1\WObj:=Workobject_2;
    SetDO Agarrar,1;
    MoveJ Target_90,v7000,fine,Mi_mecanismo_1\WObj:=Workobject_2;
    SetDO Coger_gra,1;
    SetDO Cinta_gra,1;
    SetDO Agarrar,0;
    MoveJ Target_100,v7000,fine,Mi_mecanismo_1\WObj:=Workobject_2;
    MoveJ Target_120,v7000,fine,Mi_mecanismo_1\WObj:=Workobject_2;
    MoveJ Target_130,v7000,fine,Mi_mecanismo_1\WObj:=Workobject_2;
    SetDO Coger_gra,0;
    SetDO Soltar_gra,1;
    SetDO Agarrar,1;
    MoveJ Target_120,v7000,fine,Mi_mecanismo_1\WObj:=Workobject_2;
    SetDO Agarrar,0;
    MoveJ Home,v7000,fine,Mi_mecanismo_1\WObj:=wobj0;
    SetDO Soltar_gra,0;
  ENDPROC
  PROC gra_2()
    MoveJ Home,v7000,fine,Mi_mecanismo_1\WObj:=wobj0;
    MoveJ Target_100,v7000,fine,Mi_mecanismo_1\WObj:=Workobject_2;
    SetDO Agarrar,1;
    MoveJ Target_90,v7000,fine,Mi_mecanismo_1\WObj:=Workobject_2;
    SetDO Coger_gra,1;
    SetDO Cinta_gra,1;
    SetDO Agarrar,0;
    MoveJ Target_100,v7000,fine,Mi_mecanismo_1\WObj:=Workobject_2;
    MoveJ Target_120,v7000,fine,Mi_mecanismo_1\WObj:=Workobject_2;
    MoveJ Target_140,v7000,fine,Mi_mecanismo_1\WObj:=Workobject_2;
    SetDO Coger_gra,0;
    SetDO Soltar_gra,1;
    SetDO Agarrar,1;
    MoveJ Target_120,v7000,fine,Mi_mecanismo_1\WObj:=Workobject_2;
    SetDO Agarrar,0;
    MoveJ Home,v7000,fine,Mi_mecanismo_1\WObj:=wobj0;
    SetDO Soltar_gra,0;
  ENDPROC
  PROC gra_3()
    MoveJ Home,v7000,fine,Mi_mecanismo_1\WObj:=wobj0;
    MoveJ Target_100,v7000,fine,Mi_mecanismo_1\WObj:=Workobject_2;
    SetDO Agarrar,1;
    MoveJ Target_90,v7000,fine,Mi_mecanismo_1\WObj:=Workobject_2;
    SetDO Coger_gra,1;
    SetDO Cinta_gra,1;
    SetDO Agarrar,0;
    MoveJ Target_100,v7000,fine,Mi_mecanismo_1\WObj:=Workobject_2;
    MoveJ Target_120,v7000,fine,Mi_mecanismo_1\WObj:=Workobject_2;
    MoveJ Target_150,v7000,fine,Mi_mecanismo_1\WObj:=Workobject_2;
    SetDO Coger_gra,0;
    SetDO Soltar_gra,1;
    SetDO Agarrar,1;
    MoveJ Target_120,v7000,fine,Mi_mecanismo_1\WObj:=Workobject_2;
    SetDO Agarrar,0;
    MoveJ Home,v7000,fine,Mi_mecanismo_1\WObj:=wobj0;
    SetDO Soltar_gra,0;
  ENDPROC
  PROC gra_4()
    MoveJ Home,v7000,fine,Mi_mecanismo_1\WObj:=wobj0;
    MoveJ Target_100,v7000,fine,Mi_mecanismo_1\WObj:=Workobject_2;
    SetDO Agarrar,1;
    MoveJ Target_90,v7000,fine,Mi_mecanismo_1\WObj:=Workobject_2;
    SetDO Coger_gra,1;
    SetDO Cinta_gra,1;
    SetDO Agarrar,0;
    MoveJ Target_100,v7000,fine,Mi_mecanismo_1\WObj:=Workobject_2;
    MoveJ Target_120,v7000,fine,Mi_mecanismo_1\WObj:=Workobject_2;
    MoveJ Target_160,v7000,fine,Mi_mecanismo_1\WObj:=Workobject_2;
    SetDO Coger_gra,0;
    SetDO Soltar_gra,1;
    SetDO Agarrar,1;
    MoveJ Target_120,v7000,fine,Mi_mecanismo_1\WObj:=Workobject_2;
    SetDO Agarrar,0;
    MoveJ Home,v7000,fine,Mi_mecanismo_1\WObj:=wobj0;
    SetDO Soltar_gra,0;
  ENDPROC
  PROC gra_5()
    MoveJ Home,v7000,fine,Mi_mecanismo_1\WObj:=wobj0;
    MoveJ Target_100,v7000,fine,Mi_mecanismo_1\WObj:=Workobject_2;
    SetDO Agarrar,1;
    MoveJ Target_90,v7000,fine,Mi_mecanismo_1\WObj:=Workobject_2;
    SetDO Coger_gra,1;
    SetDO Cinta_gra,1;
    SetDO Agarrar,0;
    MoveJ Target_100,v7000,fine,Mi_mecanismo_1\WObj:=Workobject_2;
    MoveJ Target_120,v7000,fine,Mi_mecanismo_1\WObj:=Workobject_2;
    MoveJ Target_170,v7000,fine,Mi_mecanismo_1\WObj:=Workobject_2;
    SetDO Coger_gra,0;
    SetDO Soltar_gra,1;
    SetDO Agarrar,1;
    MoveJ Target_120,v7000,fine,Mi_mecanismo_1\WObj:=Workobject_2;
    SetDO Agarrar,0;
    MoveJ Home,v7000,fine,Mi_mecanismo_1\WObj:=wobj0;
    SetDO Soltar_gra,0;
  ENDPROC
  PROC gra_6()
    MoveJ Home,v7000,fine,Mi_mecanismo_1\WObj:=wobj0;
    MoveJ Target_100,v7000,fine,Mi_mecanismo_1\WObj:=Workobject_2;
    SetDO Agarrar,1;
    MoveJ Target_90,v7000,fine,Mi_mecanismo_1\WObj:=Workobject_2;
    SetDO Coger_gra,1;
    SetDO Cinta_gra,1;
    SetDO Agarrar,0;
    MoveJ Target_100,v7000,fine,Mi_mecanismo_1\WObj:=Workobject_2;
    MoveJ Target_120,v7000,fine,Mi_mecanismo_1\WObj:=Workobject_2;
    MoveJ Target_180,v7000,fine,Mi_mecanismo_1\WObj:=Workobject_2;
    SetDO Coger_gra,0;
    SetDO Soltar_gra,1;
    SetDO Agarrar,1;
    MoveJ Target_120,v7000,fine,Mi_mecanismo_1\WObj:=Workobject_2;
    SetDO Agarrar,0;
    MoveJ Home,v7000,fine,Mi_mecanismo_1\WObj:=wobj0;
    SetDO Soltar_gra,0;
  ENDPROC
ENDMODULE

! task T_ROB1
MODULE pmrcUser
  TASK PERS wobjdata pmInfeeder1_WObj:=[FALSE,TRUE,"",[[0,0,0],[1,0,0,0]],[[0,0,0],[1,0,0,0]]];
  TASK PERS wobjdata pmInfeeder2_WObj:=[FALSE,TRUE,"",[[0,0,0],[1,0,0,0]],[[0,0,0],[1,0,0,0]]];
  TASK PERS wobjdata pmInfeeder3_WObj:=[FALSE,TRUE,"",[[0,0,0],[1,0,0,0]],[[0,0,0],[1,0,0,0]]];
  TASK PERS wobjdata pmInfeeder4_WObj:=[FALSE,TRUE,"",[[0,0,0],[1,0,0,0]],[[0,0,0],[1,0,0,0]]];
  TASK PERS wobjdata pmOutfeeder1_WObj:=[FALSE,TRUE,"",[[0,0,0],[1,0,0,0]],[[0,0,0],[1,0,0,0]]];
  TASK PERS wobjdata pmOutfeeder2_WObj:=[FALSE,TRUE,"",[[0,0,0],[1,0,0,0]],[[0,0,0],[1,0,0,0]]];
  TASK PERS wobjdata pmOutfeeder3_WObj:=[FALSE,TRUE,"",[[0,0,0],[1,0,0,0]],[[0,0,0],[1,0,0,0]]];
  TASK PERS wobjdata pmOutfeeder4_WObj:=[FALSE,TRUE,"",[[0,0,0],[1,0,0,0]],[[0,0,0],[1,0,0,0]]];
  TASK PERS wobjdata pmPallet1_WObj:=[FALSE,TRUE,"",[[0,0,0],[1,0,0,0]],[[0,0,0],[1,0,0,0]]];
  TASK PERS wobjdata pmSlipsheet1_WObj:=[FALSE,TRUE,"",[[0,0,0],[1,0,0,0]],[[0,0,0],[1,0,0,0]]];
  TASK PERS tooldata pmPickTool1:=[TRUE,[[0,0,0],[1,0,0,0]],[0.001,[0,0,0.001],[1,0,0,0],0,0,0]];
  TASK PERS tooldata pmSearchTool1:=[TRUE,[[0,0,0],[1,0,0,0]],[0.001,[0,0,0.001],[1,0,0,0],0,0,0]];
  TASK PERS tooldata pmCalibTool1:=[TRUE,[[0,0,0],[1,0,0,0]],[0.001,[0,0,0.001],[1,0,0,0],0,0,0]];
  PROC PmLoadReadySignalReset()
    SetDO pmSystem_doLoadReady1,0;
    SetDO pmSystem_doLoadReady2,0;
    SetDO pmSystem_doLoadReady3,0;
    SetDO pmSystem_doLoadReady4,0;
    SetDO pmSystem_doLoadReady5,0;
    SetDO pmSystem_doLoadReady6,0;
  ENDPROC
  PROC PmLoadReady()
    SetDO \Sync,pmSystem_doLoadReady1,1;
    SetDO \Sync,pmSystem_doLoadReady2,1;
    SetDO \Sync,pmSystem_doLoadReady3,1;
    SetDO \Sync,pmSystem_doLoadReady4,1;
    SetDO \Sync,pmSystem_doLoadReady5,1;
    SetDO \Sync,pmSystem_doLoadReady6,1;
  ENDPROC
  PROC PmResetProjStartFlagAtStart()
  ENDPROC
ENDMODULE

! task T_ROB1
MODULE pmrcSys
  TASK PERS wobjdata pm_home_WObj:=[FALSE,TRUE,"",[[0,0,0],[1,0,0,0]],[[0,0,0],[1,0,0,0]]];
  LOCAL PERS tooldata curr_Tool:=[TRUE,[[0,0,0],[1,0,0,0]],[0.001,[0,0,0.001],[1,0,0,0],0,0,0]];
  TASK PERS tooldata PmLastTool:=[TRUE,[[0,0,0],[1,0,0,0]],[0.001,[0,0,0.001],[1,0,0,0],0,0,0]];
  LOCAL PERS wobjdata curr_WObj:=[FALSE,TRUE,"",[[0,0,0],[1,0,0,0]],[[0,0,0],[1,0,0,0]]];
  TASK PERS wobjdata PmLastWobj:=[FALSE,TRUE,"",[[0,0,0],[1,0,0,0]],[[0,0,0],[1,0,0,0]]];
  PROC PmSetupDummyIO()
  ENDPROC
ENDMODULE

